(* IEC 61131-3 sources: rk/stdlib (part 3) *)

(* ---- Math.st ---- *)
/*
Arithmetic functions.

Each function has one overload per type it applies to, and returns the type
it was given. Angles are in radians.

A `REAL` or `LREAL` result follows IEEE 754: outside a function's domain it
is NaN, and at a pole it is infinite. Neither stops the scan. Test for them
with [Std.Math.IS_NAN] and [Std.Math.NOT_OK] where it matters.
*/
NAMESPACE Std.Math

	/* Returns the absolute value of `IN`, which is `IN` itself on an unsigned type.

	   The most negative value of a signed integer type has no positive
	   counterpart, and is returned as it is: `ABS(SINT#-128)` is -128.

	   # Examples

	   ```iecst
	   n := ABS(-5);    // 5
	   r := ABS(-2.5);  // 2.5
	   ```
	*/
	FUNCTION ABS: SINT
		VAR_INPUT
			IN: SINT
		END_VAR
		{wasm IN 'abs' (params IN) (result ABS)}
	END_FUNCTION

	FUNCTION ABS: INT
		VAR_INPUT
			IN: INT
		END_VAR
		{wasm IN 'abs' (params IN) (result ABS)}
	END_FUNCTION

	FUNCTION ABS: DINT
		VAR_INPUT
			IN: DINT
		END_VAR
		{wasm IN 'abs' (params IN) (result ABS)}
	END_FUNCTION

	FUNCTION ABS: LINT
		VAR_INPUT
			IN: LINT
		END_VAR
		{wasm IN 'abs' (params IN) (result ABS)}
	END_FUNCTION

	FUNCTION ABS: REAL
		VAR_INPUT
			IN: REAL
		END_VAR
		{wasm IN 'abs' (params IN) (result ABS)}
	END_FUNCTION

	FUNCTION ABS: LREAL
		VAR_INPUT
			IN: LREAL
		END_VAR
		{wasm IN 'abs' (params IN) (result ABS)}
	END_FUNCTION

	FUNCTION ABS: USINT
		VAR_INPUT
			IN: USINT
		END_VAR
		ABS := IN;
	END_FUNCTION

	FUNCTION ABS: UINT
		VAR_INPUT
			IN: UINT
		END_VAR
		ABS := IN;
	END_FUNCTION

	FUNCTION ABS: UDINT
		VAR_INPUT
			IN: UDINT
		END_VAR
		ABS := IN;
	END_FUNCTION

	FUNCTION ABS: ULINT
		VAR_INPUT
			IN: ULINT
		END_VAR
		ABS := IN;
	END_FUNCTION

	/* Returns the square root of `IN`.

	   Returns NaN when `IN` is negative.

	   # Examples

	   ```iecst
	   r := SQRT(9.0);  // 3.0
	   r := SQRT(2.0);  // 1.4142135
	   ```
	*/
	FUNCTION SQRT: REAL
		VAR_INPUT
			IN: REAL
		END_VAR
		{wasm IN 'sqrt' (params IN) (result SQRT)}
	END_FUNCTION

	FUNCTION SQRT: LREAL
		VAR_INPUT
			IN: LREAL
		END_VAR
		{wasm IN 'sqrt' (params IN) (result SQRT)}
	END_FUNCTION

	/* Returns the natural logarithm of `IN`.

	   Returns NaN when `IN` is negative, and negative infinity when it is 0.

	   # Examples

	   ```iecst
	   r := LN(1.0);  // 0.0
	   r := LN(2.0);  // 0.6931472
	   ```
	*/
	FUNCTION LN: REAL
		VAR_INPUT
			IN: REAL
		END_VAR
		{wasm IN 'ln' (params IN) (result LN)}
	END_FUNCTION

	FUNCTION LN: LREAL
		VAR_INPUT
			IN: LREAL
		END_VAR
		{wasm IN 'ln' (params IN) (result LN)}
	END_FUNCTION

	/* Returns the base 10 logarithm of `IN`.

	   Returns NaN when `IN` is negative, and negative infinity when it is 0.

	   # Examples

	   ```iecst
	   r := LOG(100.0);   // 2.0
	   r := LOG(1000.0);  // 3.0
	   ```
	*/
	FUNCTION LOG: REAL
		VAR_INPUT
			IN: REAL
		END_VAR
		{wasm IN 'log' (params IN) (result LOG)}
	END_FUNCTION

	FUNCTION LOG: LREAL
		VAR_INPUT
			IN: LREAL
		END_VAR
		{wasm IN 'log' (params IN) (result LOG)}
	END_FUNCTION

	/* Returns e raised to the power of `IN`.

	   # Examples

	   ```iecst
	   r := EXP(0.0);  // 1.0
	   r := EXP(1.0);  // 2.7182817
	   ```
	*/
	FUNCTION EXP: REAL
		VAR_INPUT
			IN: REAL
		END_VAR
		{wasm IN 'exp' (params IN) (result EXP)}
	END_FUNCTION

	FUNCTION EXP: LREAL
		VAR_INPUT
			IN: LREAL
		END_VAR
		{wasm IN 'exp' (params IN) (result EXP)}
	END_FUNCTION

	/* Returns the sine of `IN`, an angle in radians.

	   # Examples

	   ```iecst
	   r := SIN(0.0);  // 0.0
	   r := SIN(0.5);  // 0.4794255
	   ```
	*/
	FUNCTION SIN: REAL
		VAR_INPUT
			IN: REAL
		END_VAR
		{wasm IN 'sin' (params IN) (result SIN)}
	END_FUNCTION

	FUNCTION SIN: LREAL
		VAR_INPUT
			IN: LREAL
		END_VAR
		{wasm IN 'sin' (params IN) (result SIN)}
	END_FUNCTION

	/* Returns the cosine of `IN`, an angle in radians.

	   # Examples

	   ```iecst
	   r := COS(0.0);  // 1.0
	   r := COS(1.0);  // 0.5403023
	   ```
	*/
	FUNCTION COS: REAL
		VAR_INPUT
			IN: REAL
		END_VAR
		{wasm IN 'cos' (params IN) (result COS)}
	END_FUNCTION

	FUNCTION COS: LREAL
		VAR_INPUT
			IN: LREAL
		END_VAR
		{wasm IN 'cos' (params IN) (result COS)}
	END_FUNCTION

	/* Returns the tangent of `IN`, an angle in radians.

	   # Examples

	   ```iecst
	   r := TAN(0.0);  // 0.0
	   r := TAN(1.0);  // 1.5574077
	   ```
	*/
	FUNCTION TAN: REAL
		VAR_INPUT
			IN: REAL
		END_VAR
		{wasm IN 'tan' (params IN) (result TAN)}
	END_FUNCTION

	FUNCTION TAN: LREAL
		VAR_INPUT
			IN: LREAL
		END_VAR
		{wasm IN 'tan' (params IN) (result TAN)}
	END_FUNCTION

	/* Returns the arc sine of `IN`, in radians.

	   Returns NaN when `IN` is outside -1.0 to 1.0.

	   # Examples

	   ```iecst
	   r := ASIN(0.0);  // 0.0
	   r := ASIN(1.0);  // 1.5707964
	   ```
	*/
	FUNCTION ASIN: REAL
		VAR_INPUT
			IN: REAL
		END_VAR
		{wasm IN 'asin' (params IN) (result ASIN)}
	END_FUNCTION

	FUNCTION ASIN: LREAL
		VAR_INPUT
			IN: LREAL
		END_VAR
		{wasm IN 'asin' (params IN) (result ASIN)}
	END_FUNCTION

	/* Returns the arc cosine of `IN`, in radians.

	   Returns NaN when `IN` is outside -1.0 to 1.0.

	   # Examples

	   ```iecst
	   r := ACOS(1.0);  // 0.0
	   r := ACOS(0.0);  // 1.5707964
	   ```
	*/
	FUNCTION ACOS: REAL
		VAR_INPUT
			IN: REAL
		END_VAR
		{wasm IN 'acos' (params IN) (result ACOS)}
	END_FUNCTION

	FUNCTION ACOS: LREAL
		VAR_INPUT
			IN: LREAL
		END_VAR
		{wasm IN 'acos' (params IN) (result ACOS)}
	END_FUNCTION

	/* Returns the arc tangent of `IN`, in radians.

	   # Examples

	   ```iecst
	   r := ATAN(0.0);  // 0.0
	   r := ATAN(1.0);  // 0.7853982
	   ```
	*/
	FUNCTION ATAN: REAL
		VAR_INPUT
			IN: REAL
		END_VAR
		{wasm IN 'atan' (params IN) (result ATAN)}
	END_FUNCTION

	FUNCTION ATAN: LREAL
		VAR_INPUT
			IN: LREAL
		END_VAR
		{wasm IN 'atan' (params IN) (result ATAN)}
	END_FUNCTION

	/* Returns the angle of the point (`X`, `Y`), in radians.

	   This is the arc tangent of `IN / IN2`, with the signs of both used to pick
	   the quadrant. `Y` is the y coordinate and `X` the x.

	   # Examples

	   ```iecst
	   r := ATAN2(1.0, 1.0);    // 0.7853982
	   r := ATAN2(1.0, -1.0);   // 2.3561945
	   r := ATAN2(-1.0, 1.0);   // -0.7853982
	   ```
	*/
	FUNCTION ATAN2: REAL
		VAR_INPUT
			Y: REAL
			X: REAL
		END_VAR
		{wasm Y 'atan2' (params Y X) (result ATAN2)}
	END_FUNCTION

	FUNCTION ATAN2: LREAL
		VAR_INPUT
			Y: LREAL
			X: LREAL
		END_VAR
		{wasm Y 'atan2' (params Y X) (result ATAN2)}
	END_FUNCTION

	/* Returns `IN1` raised to the power of `IN2`.

	   This is the `**` operator as a function. `IN2` may be an integer, and the
	   result has the type of `IN1`.

	   # Examples

	   ```iecst
	   r := EXPT(2.0, 3.0);  // 8.0
	   r := EXPT(9.0, 0.5);  // 3.0
	   ```
	*/
	FUNCTION EXPT: REAL
		VAR_INPUT
			IN1: REAL
			IN2: REAL
		END_VAR
		{wasm IN1 'pow' (params IN1 IN2) (result EXPT)}
	END_FUNCTION

	FUNCTION EXPT: LREAL
		VAR_INPUT
			IN1: LREAL
			IN2: LREAL
		END_VAR
		{wasm IN1 'pow' (params IN1 IN2) (result EXPT)}
	END_FUNCTION

	FUNCTION EXPT: REAL
		VAR_INPUT
			IN1: REAL
			IN2: LREAL
		END_VAR
		EXPT := IN1 ** IN2;
	END_FUNCTION

	FUNCTION EXPT: REAL
		VAR_INPUT
			IN1: REAL
			IN2: SINT
		END_VAR
		EXPT := IN1 ** IN2;
	END_FUNCTION

	FUNCTION EXPT: REAL
		VAR_INPUT
			IN1: REAL
			IN2: INT
		END_VAR
		EXPT := IN1 ** IN2;
	END_FUNCTION

	FUNCTION EXPT: REAL
		VAR_INPUT
			IN1: REAL
			IN2: DINT
		END_VAR
		EXPT := IN1 ** IN2;
	END_FUNCTION

	FUNCTION EXPT: REAL
		VAR_INPUT
			IN1: REAL
			IN2: LINT
		END_VAR
		EXPT := IN1 ** IN2;
	END_FUNCTION

	FUNCTION EXPT: REAL
		VAR_INPUT
			IN1: REAL
			IN2: USINT
		END_VAR
		EXPT := IN1 ** IN2;
	END_FUNCTION

	FUNCTION EXPT: REAL
		VAR_INPUT
			IN1: REAL
			IN2: UINT
		END_VAR
		EXPT := IN1 ** IN2;
	END_FUNCTION

	FUNCTION EXPT: REAL
		VAR_INPUT
			IN1: REAL
			IN2: UDINT
		END_VAR
		EXPT := IN1 ** IN2;
	END_FUNCTION

	FUNCTION EXPT: REAL
		VAR_INPUT
			IN1: REAL
			IN2: ULINT
		END_VAR
		EXPT := IN1 ** IN2;
	END_FUNCTION

	FUNCTION EXPT: LREAL
		VAR_INPUT
			IN1: LREAL
			IN2: REAL
		END_VAR
		EXPT := IN1 ** IN2;
	END_FUNCTION

	FUNCTION EXPT: LREAL
		VAR_INPUT
			IN1: LREAL
			IN2: SINT
		END_VAR
		EXPT := IN1 ** IN2;
	END_FUNCTION

	FUNCTION EXPT: LREAL
		VAR_INPUT
			IN1: LREAL
			IN2: INT
		END_VAR
		EXPT := IN1 ** IN2;
	END_FUNCTION

	FUNCTION EXPT: LREAL
		VAR_INPUT
			IN1: LREAL
			IN2: DINT
		END_VAR
		EXPT := IN1 ** IN2;
	END_FUNCTION

	FUNCTION EXPT: LREAL
		VAR_INPUT
			IN1: LREAL
			IN2: LINT
		END_VAR
		EXPT := IN1 ** IN2;
	END_FUNCTION

	FUNCTION EXPT: LREAL
		VAR_INPUT
			IN1: LREAL
			IN2: USINT
		END_VAR
		EXPT := IN1 ** IN2;
	END_FUNCTION

	FUNCTION EXPT: LREAL
		VAR_INPUT
			IN1: LREAL
			IN2: UINT
		END_VAR
		EXPT := IN1 ** IN2;
	END_FUNCTION

	FUNCTION EXPT: LREAL
		VAR_INPUT
			IN1: LREAL
			IN2: UDINT
		END_VAR
		EXPT := IN1 ** IN2;
	END_FUNCTION

	FUNCTION EXPT: LREAL
		VAR_INPUT
			IN1: LREAL
			IN2: ULINT
		END_VAR
		EXPT := IN1 ** IN2;
	END_FUNCTION

	/* Returns `TRUE` if `IN` is not a number.

	   NaN comes from `0.0 / 0.0`, from the square root of a negative, and above
	   all from a bit pattern read off a fieldbus or an analog channel. It spreads
	   through arithmetic and converts to 0, so test for it where it matters.

	   See [Std.Math.NOT_OK] to refuse an infinite value as well.
	*/
	FUNCTION IS_NAN: BOOL
		VAR_INPUT
			IN: REAL;
		END_VAR
		IS_NAN := IN <> IN;
	END_FUNCTION

	FUNCTION IS_NAN: BOOL
		VAR_INPUT
			IN: LREAL;
		END_VAR
		IS_NAN := IN <> IN;
	END_FUNCTION

	/* Returns `TRUE` if `IN` is not a number, or is infinite.

	   # Examples

	   ```iecst
	   IF NOT_OK(measured) THEN
	       alarm := TRUE;
	   END_IF;
	   ```
	*/
	FUNCTION NOT_OK: BOOL
		VAR_INPUT
			IN: REAL;
		END_VAR
		NOT_OK := (IN - IN) <> 0.0;
	END_FUNCTION

	FUNCTION NOT_OK: BOOL
		VAR_INPUT
			IN: LREAL;
		END_VAR
		NOT_OK := (IN - IN) <> LREAL#0.0;
	END_FUNCTION

	NAMESPACE Test
		USING Std.Unit

		// ----- EXPT ---------------------------------------------------
		{test}
		FUNCTION test_is_nan
			VAR
				z: REAL := 0.0;
			END_VAR
			ASSERT(IS_NAN(z / z) AND NOT IS_NAN(1.5) AND NOT IS_NAN(1.0 / z));
		END_FUNCTION

		{test}
		FUNCTION test_not_ok_is_nan_or_infinite
			VAR
				z: REAL := 0.0;
			END_VAR
			ASSERT(NOT_OK(z / z) AND NOT_OK(1.0 / z) AND NOT_OK(-1.0 / z) AND NOT NOT_OK(3.0));
		END_FUNCTION

		{test}
		FUNCTION test_expt_real ASSERT(EXPT(2.0, 3.0) = 8.0);
		END_FUNCTION

		{test}
		FUNCTION test_expt_fractional ASSERT(EXPT(9.0, 0.5) = 3.0);
		END_FUNCTION

		// The result has the type of IN1, whatever the exponent's: a REAL
		// raised to a DINT is stored in a REAL, which an LREAL result is not.
		{test}
		FUNCTION test_expt_keeps_the_base_type
		VAR r: REAL; l: LREAL; n: DINT := 3; u: USINT := 10; END_VAR
			r := EXPT(REAL#2.0, n);
			ASSERT(r = 8.0);
			r := EXPT(REAL#2.0, LREAL#0.5);
			ASSERT(r > 1.41 AND r < 1.42);
			l := EXPT(LREAL#2.0, u);
			ASSERT(l = LREAL#1024.0);
		END_FUNCTION

		{test}
		FUNCTION test_expt_integer_exponent
		VAR x: REAL; n: INT; END_VAR
			x := 2.0;
			n := 10;
			ASSERT(EXPT(x, n) = 1024.0);
		END_FUNCTION

		{test}
		FUNCTION test_expt_lreal ASSERT(EXPT(LREAL#2.0, LREAL#10.0) = LREAL#1024.0);
		END_FUNCTION

		// The result has the type of IN1, whatever the exponent: a REAL target
		// refuses an LREAL.
		{test}
		FUNCTION test_expt_keeps_the_type_of_in1
			VAR
				r: REAL := 2.0;
				l: LREAL := 2.0;
				a: REAL;
				b: LREAL;
				si: SINT := 3;
				i: INT := 3;
				d: DINT := 3;
				n: LINT := 3;
				us: USINT := 3;
				u: UINT := 3;
				ud: UDINT := 3;
				ul: ULINT := 3;
				x: REAL := 3.0;
				y: LREAL := 3.0;
			END_VAR
			a := EXPT(r, si); ASSERT(a = 8.0);
			a := EXPT(r, i); ASSERT(a = 8.0);
			a := EXPT(r, d); ASSERT(a = 8.0);
			a := EXPT(r, n); ASSERT(a = 8.0);
			a := EXPT(r, us); ASSERT(a = 8.0);
			a := EXPT(r, u); ASSERT(a = 8.0);
			a := EXPT(r, ud); ASSERT(a = 8.0);
			a := EXPT(r, ul); ASSERT(a = 8.0);
			a := EXPT(r, x); ASSERT(a = 8.0);
			a := EXPT(r, y); ASSERT(a = 8.0);
			b := EXPT(l, si); ASSERT(b = LREAL#8.0);
			b := EXPT(l, i); ASSERT(b = LREAL#8.0);
			b := EXPT(l, d); ASSERT(b = LREAL#8.0);
			b := EXPT(l, n); ASSERT(b = LREAL#8.0);
			b := EXPT(l, us); ASSERT(b = LREAL#8.0);
			b := EXPT(l, u); ASSERT(b = LREAL#8.0);
			b := EXPT(l, ud); ASSERT(b = LREAL#8.0);
			b := EXPT(l, ul); ASSERT(b = LREAL#8.0);
			b := EXPT(l, x); ASSERT(b = LREAL#8.0);
			b := EXPT(l, y); ASSERT(b = LREAL#8.0);
		END_FUNCTION

		{test}
		FUNCTION test_expt_takes_literals
			VAR
				r: REAL := 2.0;
				l: LREAL := 2.0;
				a: REAL;
				b: LREAL;
			END_VAR
			a := EXPT(2.0, 3.0); ASSERT(a = 8.0);
			a := EXPT(r, 3.0); ASSERT(a = 8.0);
			a := EXPT(r, 3); ASSERT(a = 8.0);
			a := EXPT(2.0, 3); ASSERT(a = 8.0);
			a := EXPT(r, DINT#3); ASSERT(a = 8.0);
			a := EXPT(IN1 := r, IN2 := 3); ASSERT(a = 8.0);
			b := EXPT(l, 3); ASSERT(b = LREAL#8.0);
			b := EXPT(l, 3.0); ASSERT(b = LREAL#8.0);
			b := EXPT(LREAL#2.0, 3); ASSERT(b = LREAL#8.0);
			b := EXPT(l, -1); ASSERT(b = LREAL#0.5);
		END_FUNCTION

		{test}
		FUNCTION test_abs_of_an_unsigned_is_itself
			VAR
				us: USINT := 200;
				u: UINT := 60000;
				ud: UDINT := 4000000000;
				ul: ULINT := 18446744073709551615;
			END_VAR
			us := ABS(us); ASSERT(us = 200);
			u := ABS(u); ASSERT(u = 60000);
			ud := ABS(ud); ASSERT(ud = 4000000000);
			ul := ABS(ul); ASSERT(ul = 18446744073709551615);
		END_FUNCTION

		{test}
		FUNCTION test_expt_matches_operator
		VAR x: REAL; END_VAR
			x := 3.0;
			ASSERT(EXPT(x, 2.0) = x ** 2.0);
		END_FUNCTION

		// ----- ABS (per signed-numeric overloads) ---------------------
		{test}
		FUNCTION test_abs_positive ASSERT(ABS(5) = 5);
		END_FUNCTION

		{test}
		FUNCTION test_abs_negative ASSERT(ABS(-42) = 42);
		END_FUNCTION

		{test}
		FUNCTION test_abs_zero ASSERT(ABS(0) = 0);
		END_FUNCTION

		{test}
		FUNCTION test_abs_real ASSERT(ABS(-2.5) = 2.5);
		END_FUNCTION

		{test}
		FUNCTION test_abs_real_positive ASSERT(ABS(3.14) = 3.14);
		END_FUNCTION

		{test}
		FUNCTION test_abs_with_message ASSERT(ABS(-7) = 7, 'ABS should return the positive value');
		END_FUNCTION

		// An unsigned value is its own absolute value, the largest included.
		{test}
		FUNCTION test_abs_unsigned
			ASSERT(ABS(USINT#255) = USINT#255);
			ASSERT(ABS(UINT#65535) = UINT#65535);
			ASSERT(ABS(UDINT#4294967295) = UDINT#4294967295);
			ASSERT(ABS(ULINT#18446744073709551615) = ULINT#18446744073709551615);
		END_FUNCTION

		// ----- SQRT (REAL/LREAL overloads) ----------------------------
		{test}
		FUNCTION test_sqrt_9 ASSERT(SQRT(9.0) = 3.0);
		END_FUNCTION

		{test}
		FUNCTION test_sqrt_4 ASSERT(SQRT(4.0) = 2.0);
		END_FUNCTION

		{test}
		FUNCTION test_sqrt_1 ASSERT(SQRT(1.0) = 1.0);
		END_FUNCTION

		// ----- Trigonometric (REAL/LREAL overloads) -------------------
		{test}
		FUNCTION test_sin_zero ASSERT(SIN(0.0) = 0.0);
		END_FUNCTION

		{test}
		FUNCTION test_cos_zero ASSERT(COS(0.0) = 1.0);
		END_FUNCTION

		{test}
		FUNCTION test_tan_zero ASSERT(TAN(0.0) = 0.0);
		END_FUNCTION

		{test}
		FUNCTION test_asin_zero ASSERT(ASIN(0.0) = 0.0);
		END_FUNCTION

		{test}
		FUNCTION test_acos_one ASSERT(ACOS(1.0) = 0.0);
		END_FUNCTION

		{test}
		FUNCTION test_atan_zero ASSERT(ATAN(0.0) = 0.0);
		END_FUNCTION

		// ----- Logarithmic / Exponential (REAL/LREAL overloads) ------
		{test}
		FUNCTION test_ln_1 ASSERT(LN(1.0) = 0.0);
		END_FUNCTION

		{test}
		FUNCTION test_log_1 ASSERT(LOG(1.0) = 0.0);
		END_FUNCTION

		{test}
		FUNCTION test_exp_0 ASSERT(EXP(0.0) = 1.0);
		END_FUNCTION

		// ----- Arithmetic operators --------------------------------------------------------------------------------
		{test}
		FUNCTION test_add_int
			VAR
				r: INT;
			END_VAR
			r := 3 + 4;
			ASSERT(r = 7);
		END_FUNCTION

		{test}
		FUNCTION test_sub_int
			VAR
				r: INT;
			END_VAR
			r := 10 - 3;
			ASSERT(r = 7);
		END_FUNCTION

		{test}
		FUNCTION test_mul_int
			VAR
				r: INT;
			END_VAR
			r := 6 * 7;
			ASSERT(r = 42);
		END_FUNCTION

		{test}
		FUNCTION test_div_int
			VAR
				r: INT;
			END_VAR
			r := 100 / 10;
			ASSERT(r = 10);
		END_FUNCTION

		{test}
		FUNCTION test_mod_int
			VAR
				r: INT;
			END_VAR
			r := 10 MOD 3;
			ASSERT(r = 1);
		END_FUNCTION

		{test}
		FUNCTION test_add_real
			VAR
				r: REAL;
			END_VAR
			r := 1.5 + 2.5;
			ASSERT(r = 4.0);
		END_FUNCTION

		{test}
		FUNCTION test_sub_negative
			VAR
				r: INT;
			END_VAR
			r := 3 - 10;
			ASSERT(r = -7);
		END_FUNCTION

		{test}
		FUNCTION test_nested_arithmetic
			VAR
				a: INT;
				b: INT;
				c: INT;
			END_VAR
			a := 2 * 3;
			b := 4 * 5;
			c := a + b;
			ASSERT(c = 26);
		END_FUNCTION

		// ----- Variable assignment ---------------------------------------------------------------------------------
		{test}
		FUNCTION test_var_assignment
			VAR
				x: INT := 10;
				y: INT;
			END_VAR
			y := x;
			ASSERT(x = y);
		END_FUNCTION

		{test}
		FUNCTION test_var_init
			VAR
				x: INT := 42;
			END_VAR
			ASSERT(x = 42);
		END_FUNCTION

		{test}
		FUNCTION test_var_default_zero
			VAR
				x: INT;
			END_VAR
			ASSERT(x = 0);
		END_FUNCTION

		{test}
		FUNCTION test_var_bool_init
			VAR
				b: BOOL := TRUE;
			END_VAR
			ASSERT(b);
		END_FUNCTION

		{test}
		FUNCTION test_var_real_init
			VAR
				r: REAL := 3.14;
			END_VAR
			ASSERT(r = 3.14);
		END_FUNCTION

		// ----- Boolean logic ---------------------------------------------------------------------------------------
		{test}
		FUNCTION test_bool_and_tt
			VAR
				a: BOOL := TRUE;
				b: BOOL := TRUE;
			END_VAR
			ASSERT(a AND b);
		END_FUNCTION

		{test}
		FUNCTION test_bool_and_tf
			VAR
				a: BOOL := TRUE;
				b: BOOL := FALSE;
			END_VAR
			ASSERT(NOT (a AND b));
		END_FUNCTION

		{test}
		FUNCTION test_bool_or_tf
			VAR
				a: BOOL := FALSE;
				b: BOOL := TRUE;
			END_VAR
			ASSERT(a OR b);
		END_FUNCTION

		{test}
		FUNCTION test_bool_or_ff
			VAR
				a: BOOL := FALSE;
				b: BOOL := FALSE;
			END_VAR
			ASSERT(NOT (a OR b));
		END_FUNCTION

		{test}
		FUNCTION test_bool_not
			VAR
				a: BOOL := FALSE;
			END_VAR
			ASSERT(NOT a);
		END_FUNCTION

		{test}
		FUNCTION test_bool_xor
			VAR
				a: BOOL := TRUE;
				b: BOOL := FALSE;
			END_VAR
			ASSERT(a XOR b);
		END_FUNCTION

		{test}
		FUNCTION test_bool_xor_same
			VAR
				a: BOOL := TRUE;
				b: BOOL := TRUE;
			END_VAR
			ASSERT(NOT (a XOR b));
		END_FUNCTION

		// ----- Comparison operators --------------------------------------------------------------------------------
		{test}
		FUNCTION test_cmp_eq
			VAR
				a: INT := 5;
			END_VAR
			ASSERT(a = 5);
		END_FUNCTION

		{test}
		FUNCTION test_cmp_ne
			VAR
				a: INT := 1;
				b: INT := 2;
			END_VAR
			ASSERT(a <> b);
		END_FUNCTION

		{test}
		FUNCTION test_cmp_lt
			VAR
				a: INT := 3;
				b: INT := 5;
			END_VAR
			ASSERT(a < b);
		END_FUNCTION

		{test}
		FUNCTION test_cmp_le
			VAR
				a: INT := 5;
			END_VAR
			ASSERT(a <= 5);
		END_FUNCTION

		{test}
		FUNCTION test_cmp_gt
			VAR
				a: INT := 10;
				b: INT := 5;
			END_VAR
			ASSERT(a > b);
		END_FUNCTION

		{test}
		FUNCTION test_cmp_ge
			VAR
				a: INT := 5;
			END_VAR
			ASSERT(a >= 5);
		END_FUNCTION

		// ----- Control flow: IF ------------------------------------------------------------------------------------
		{test}
		FUNCTION test_if_true
			VAR
				r: INT := 0;
			END_VAR
			IF TRUE THEN
				r := 1;
			END_IF;
			ASSERT(r = 1);
		END_FUNCTION

		{test}
		FUNCTION test_if_false
			VAR
				r: INT := 0;
			END_VAR
			IF FALSE THEN
				r := 1;
			END_IF;
			ASSERT(r = 0);
		END_FUNCTION

		{test}
		FUNCTION test_if_else
			VAR
				r: INT := 0;
			END_VAR
			IF FALSE THEN
				r := 1;
			ELSE
				r := 2;
			END_IF;
			ASSERT(r = 2);
		END_FUNCTION

		{test}
		FUNCTION test_if_elsif
			VAR
				r: INT := 0;
				x: INT := 2;
			END_VAR
			IF x = 1 THEN
				r := 10;
			ELSIF x = 2 THEN
				r := 20;
			ELSE
				r := 30;
			END_IF;
			ASSERT(r = 20);
		END_FUNCTION

		// ----- Control flow: FOR -----------------------------------------------------------------------------------
		{test}
		FUNCTION test_for_sum
			VAR
				sum: INT := 0;
				i: INT;
			END_VAR
			FOR i := 1 TO 5 DO
				sum := sum + i;
			END_FOR;
			ASSERT(sum = 15);
		END_FUNCTION

		{test}
		FUNCTION test_for_single
			VAR
				r: INT := 0;
				i: INT;
			END_VAR
			FOR i := 5 TO 5 DO
				r := r + 1;
			END_FOR;
			ASSERT(r = 1);
		END_FUNCTION

		{test}
		FUNCTION test_for_descending
			VAR
				n: INT := 0;
				i: INT;
			END_VAR
			// A constant negative BY flips the exit comparison: this loop
			// used to exit before its first iteration.
			FOR i := 10 TO 1 BY -1 DO
				n := n + 1;
			END_FOR;
			ASSERT(n = 10, 'descending FOR runs all 10 iterations');
		END_FUNCTION

		{test}
		FUNCTION test_for_lint_counter
			VAR
				n: LINT := 0;
				i: LINT;
			END_VAR
			// i64-lane control variable (used to emit invalid wasm).
			FOR i := LINT#1 TO LINT#3 DO
				n := n + i;
			END_FOR;
			ASSERT(n = LINT#6, 'LINT FOR loop sums 1+2+3');
		END_FUNCTION

		{test}
		FUNCTION test_for_lint_descending_beyond_i32
			VAR
				n: LINT := 0;
				i: LINT;
			END_VAR
			FOR i := LINT#5000000002 TO LINT#5000000000 BY LINT#-1 DO
				n := n + 1;
			END_FOR;
			ASSERT(n = LINT#3, 'descending i64 FOR with bounds beyond i32 range');
		END_FUNCTION

		{test}
		FUNCTION test_for_subwidth_counter_stays_in_domain
			VAR
				n: USINT := 0;
				i: USINT;
			END_VAR
			// Counter increments stay in the type's domain. NOTE: an upper
			// bound at the type MAX (e.g. TO 255) wraps before the exit
			// check and never terminates; keep bounds below the type maximum.
			FOR i := 250 TO 254 DO
				n := n + 1;
			END_FOR;
			ASSERT(n = USINT#5, 'body ran 5 times');
			{allow 'loop-var-after-loop'}
			ASSERT(i = USINT#255, 'counter exits in-domain at 255');
		END_FUNCTION

		// ----- Control flow: WHILE ---------------------------------------------------------------------------------
		{test}
		FUNCTION test_while_count
			VAR
				count: INT := 0;
			END_VAR
			WHILE count < 10 DO
				count := count + 1;
			END_WHILE;
			ASSERT(count = 10);
		END_FUNCTION

		{test}
		FUNCTION test_while_false
			VAR
				count: INT := 0;
			END_VAR
			WHILE FALSE DO
				count := count + 1;
			END_WHILE;
			ASSERT(count = 0);
		END_FUNCTION

		// ----- Control flow: REPEAT --------------------------------------------------------------------------------
		{test}
		FUNCTION test_repeat_until
			VAR
				count: INT := 0;
			END_VAR
			REPEAT count := count + 1;
				UNTIL count >= 5
			END_REPEAT;
			ASSERT(count = 5);
		END_FUNCTION

		// ----- Function calls with return values ----------------------
		{test}
		FUNCTION test_func_return
			VAR
				r: INT;
			END_VAR
			r := ABS(-99);
			ASSERT(r = 99);
		END_FUNCTION

		// Chained calls via intermediate variable
		{test}
		FUNCTION test_chained_abs
			VAR
				inner: INT;
				r: INT;
			END_VAR
			inner := ABS(-5);
			r := ABS(inner);
			ASSERT(r = 5);
		END_FUNCTION

		// ----- Type widths -----------------------------------------------------------------------------------------
		{test}
		FUNCTION test_lint_arithmetic
			VAR
				a: LINT := 1000000000;
				b: LINT := 2000000000;
				c: LINT;
			END_VAR
			c := a + b;
			ASSERT(c = 3000000000);
		END_FUNCTION

		{test}
		FUNCTION test_lreal_precision
			VAR
				a: LREAL := 1.0;
				b: LREAL := 3.0;
				c: LREAL;
			END_VAR
			c := a / b;
			// Can't compare exactly, but c * 3.0 should be 1.0
			ASSERT(c * b = a);
		END_FUNCTION

		// --- transcendentals at nonzero, non-colliding points: the fixed
		// points used above (0->0, 1->0, 0->1) are shared across the whole
		// family, so swapped imports (ln vs log, exp vs cos) pass unnoticed ---

		{test}
		FUNCTION test_trig_nonzero_points_real
			ASSERT(ABS(SIN(0.5) - 0.4794255) < 0.0001, 'SIN(0.5)');
			ASSERT(ABS(COS(1.0) - 0.5403023) < 0.0001, 'COS(1.0)');
			ASSERT(ABS(TAN(1.0) - 1.5574077) < 0.0001, 'TAN(1.0)');
			ASSERT(ABS(ASIN(0.5) - 0.5235988) < 0.0001, 'ASIN(0.5) = pi/6');
			ASSERT(ABS(ACOS(0.5) - 1.0471976) < 0.0001, 'ACOS(0.5) = pi/3');
			ASSERT(ABS(ATAN(1.0) - 0.7853982) < 0.0001, 'ATAN(1.0) = pi/4');
		END_FUNCTION

		{test}
		FUNCTION test_trig_nonzero_points_lreal
			ASSERT(ABS(SIN(LREAL#0.5) - LREAL#0.479425538604203) < LREAL#0.000000001, 'SIN LREAL');
			ASSERT(ABS(COS(LREAL#1.0) - LREAL#0.540302305868140) < LREAL#0.000000001, 'COS LREAL');
			ASSERT(ABS(ATAN(LREAL#1.0) - LREAL#0.785398163397448) < LREAL#0.000000001, 'ATAN LREAL = pi/4');
		END_FUNCTION

		{test}
		FUNCTION test_log_exp_nonzero_points
			ASSERT(ABS(LN(2.0) - 0.6931472) < 0.0001, 'LN(2)');
			ASSERT(ABS(LOG(100.0) - 2.0) < 0.0001, 'LOG(100) = 2, distinguishes LOG from LN');
			ASSERT(ABS(EXP(1.0) - 2.7182818) < 0.0001, 'EXP(1) = e');
			ASSERT(ABS(SQRT(2.0) - 1.4142136) < 0.0001, 'SQRT(2)');
			ASSERT(ABS(LN(LREAL#2.0) - LREAL#0.693147180559945) < LREAL#0.000000001, 'LN LREAL');
			ASSERT(ABS(EXP(LREAL#1.0) - LREAL#2.718281828459045) < LREAL#0.000000001, 'EXP LREAL');
			ASSERT(ABS(LOG(LREAL#1000.0) - LREAL#3.0) < LREAL#0.000000001, 'LOG LREAL');
			ASSERT(ABS(SQRT(LREAL#2.0) - LREAL#1.414213562373095) < LREAL#0.000000001, 'SQRT LREAL');
		END_FUNCTION

		// --- ATAN2: the one two-argument function. Swapped y/x is only
		// detectable with an asymmetric quadrant pair ---

		{test}
		FUNCTION test_atan2_quadrants_real
			ASSERT(ABS(ATAN2(1.0, -1.0) - 2.3561945) < 0.0001, 'ATAN2(+y,-x) = 3pi/4 (2nd quadrant)');
			ASSERT(ABS(ATAN2(-1.0, 1.0) - (-0.7853982)) < 0.0001, 'ATAN2(-y,+x) = -pi/4 (4th quadrant)');
		END_FUNCTION

		{test}
		FUNCTION test_atan2_quadrants_lreal
			ASSERT(ABS(ATAN2(LREAL#1.0, LREAL#-1.0) - LREAL#2.356194490192345) < LREAL#0.000000001, 'ATAN2 LREAL 3pi/4');
			ASSERT(ABS(ATAN2(LREAL#-1.0, LREAL#1.0) - LREAL#-0.785398163397448) < LREAL#0.000000001, 'ATAN2 LREAL -pi/4');
		END_FUNCTION

		// --- ABS boundaries and the dark overloads ---

		{test}
		FUNCTION test_abs_boundaries
			ASSERT_EQ(ABS(SINT#-127), SINT#127, 'ABS SINT near MIN');
			ASSERT_EQ(ABS(INT#-32767), INT#32767, 'ABS INT near MIN');
			ASSERT_EQ(ABS(DINT#-2147483647), DINT#2147483647, 'ABS DINT near MIN');
			ASSERT_EQ(ABS(LINT#-5000000000), LINT#5000000000, 'ABS LINT on the i64 lane');
		END_FUNCTION

		// --- sub-width integer arithmetic wraps at the IEC type width.
		// Values must never escape the type's domain ---

		{test}
		FUNCTION test_subwidth_arithmetic_wraps
			VAR
				a: USINT := 255;
				b: USINT := 1;
				z: USINT := 0;
				m: USINT := 16;
				i: INT := 32767;
				one: INT := 1;
				imin: INT := -32768;
				u16a: UINT := 65535;
			END_VAR
			ASSERT(a + b = USINT#0, 'USINT 255+1 wraps to 0');
			ASSERT(z - b = USINT#255, 'USINT 0-1 wraps to 255');
			ASSERT(m * m = USINT#0, 'USINT 16*16 wraps to 0');
			ASSERT(i + one = INT#-32768, 'INT 32767+1 wraps to -32768');
			ASSERT(imin - one = INT#32767, 'INT -32768-1 wraps to 32767');
			ASSERT(u16a * u16a = UINT#1, 'UINT 65535*65535 wraps to 1');
		END_FUNCTION

		{test}
		FUNCTION test_subwidth_negation_wraps
			VAR
				s: SINT := -128;
				sm1: SINT := -1;
			END_VAR
			ASSERT(-s = SINT#-128, 'NEG(SINT#-128) wraps to -128');
			ASSERT(s / sm1 = SINT#-128, 'SINT -128/-1 wraps to -128');
			ASSERT(ABS(s) = SINT#-128, 'ABS(SINT#-128) wraps to -128');
			ASSERT(ABS(SINT#-127) = SINT#127, 'ABS in-range is unaffected');
		END_FUNCTION

		// --- domain edges (pins current IEEE 754 behavior through libm) ---

		{test}
		FUNCTION test_float_domain_edges_pin_current
			(* pins current behavior: IEEE semantics, NaN for out-of-domain,
			   infinities at the poles. NaN is the only value with x <> x. *)
			ASSERT(SQRT(-1.0) <> SQRT(-1.0), 'SQRT(-1) is NaN');
			ASSERT(LN(-1.0) <> LN(-1.0), 'LN(-1) is NaN');
			ASSERT(LN(0.0) < -1000000.0, 'LN(0) is -inf');
			ASSERT(EXP(1000.0) > 1000000.0, 'EXP(1000) overflows to +inf');
		END_FUNCTION

		// wasm traps on the minimum divided by -1; the compiler guards it, so
		// the quotient wraps like every other overflow.
		{test}
		FUNCTION test_division_at_the_minimum_wraps
			VAR i : INT := INT#-32768; d : DINT := DINT#-2147483648; l : LINT := -LINT#9223372036854775807 - LINT#1; END_VAR
			ASSERT(i / INT#-1 = INT#-32768, 'INT');
			ASSERT(d / DINT#-1 = DINT#-2147483648, 'DINT');
			ASSERT(l / LINT#-1 = l, 'LINT');
			ASSERT(d MOD DINT#-1 = DINT#0, 'MOD is 0');
		END_FUNCTION
	END_NAMESPACE
END_NAMESPACE

(* ---- Memory.st ---- *)
/*
Memory functions.
*/
NAMESPACE Std.Memory

	/* Returns `IN`, and copies it into `OUT`.

	   There is one overload per elementary type.

	   # Examples

	   ```iecst
	   x := MOVE(42);       // x is 42
	   MOVE(42, OUT => x);  // x is 42
	   ```
	*/
	FUNCTION MOVE: BOOL
		VAR_INPUT
			IN: BOOL;
		END_VAR
		VAR_OUTPUT
			OUT: BOOL;
		END_VAR

		OUT := IN;
		MOVE := IN;
	END_FUNCTION

	FUNCTION MOVE: SINT
		VAR_INPUT
			IN: SINT;
		END_VAR
		VAR_OUTPUT
			OUT: SINT;
		END_VAR

		OUT := IN;
		MOVE := IN;
	END_FUNCTION

	FUNCTION MOVE: INT
		VAR_INPUT
			IN: INT;
		END_VAR
		VAR_OUTPUT
			OUT: INT;
		END_VAR

		OUT := IN;
		MOVE := IN;
	END_FUNCTION

	FUNCTION MOVE: DINT
		VAR_INPUT
			IN: DINT;
		END_VAR
		VAR_OUTPUT
			OUT: DINT;
		END_VAR

		OUT := IN;
		MOVE := IN;
	END_FUNCTION

	FUNCTION MOVE: LINT
		VAR_INPUT
			IN: LINT;
		END_VAR
		VAR_OUTPUT
			OUT: LINT;
		END_VAR

		OUT := IN;
		MOVE := IN;
	END_FUNCTION

	FUNCTION MOVE: USINT
		VAR_INPUT
			IN: USINT;
		END_VAR
		VAR_OUTPUT
			OUT: USINT;
		END_VAR

		OUT := IN;
		MOVE := IN;
	END_FUNCTION

	FUNCTION MOVE: UINT
		VAR_INPUT
			IN: UINT;
		END_VAR
		VAR_OUTPUT
			OUT: UINT;
		END_VAR

		OUT := IN;
		MOVE := IN;
	END_FUNCTION

	FUNCTION MOVE: UDINT
		VAR_INPUT
			IN: UDINT;
		END_VAR
		VAR_OUTPUT
			OUT: UDINT;
		END_VAR

		OUT := IN;
		MOVE := IN;
	END_FUNCTION

	FUNCTION MOVE: ULINT
		VAR_INPUT
			IN: ULINT;
		END_VAR
		VAR_OUTPUT
			OUT: ULINT;
		END_VAR

		OUT := IN;
		MOVE := IN;
	END_FUNCTION

	FUNCTION MOVE: BYTE
		VAR_INPUT
			IN: BYTE;
		END_VAR
		VAR_OUTPUT
			OUT: BYTE;
		END_VAR

		OUT := IN;
		MOVE := IN;
	END_FUNCTION

	FUNCTION MOVE: WORD
		VAR_INPUT
			IN: WORD;
		END_VAR
		VAR_OUTPUT
			OUT: WORD;
		END_VAR

		OUT := IN;
		MOVE := IN;
	END_FUNCTION

	FUNCTION MOVE: DWORD
		VAR_INPUT
			IN: DWORD;
		END_VAR
		VAR_OUTPUT
			OUT: DWORD;
		END_VAR

		OUT := IN;
		MOVE := IN;
	END_FUNCTION

	FUNCTION MOVE: LWORD
		VAR_INPUT
			IN: LWORD;
		END_VAR
		VAR_OUTPUT
			OUT: LWORD;
		END_VAR

		OUT := IN;
		MOVE := IN;
	END_FUNCTION

	FUNCTION MOVE: REAL
		VAR_INPUT
			IN: REAL;
		END_VAR
		VAR_OUTPUT
			OUT: REAL;
		END_VAR

		OUT := IN;
		MOVE := IN;
	END_FUNCTION

	FUNCTION MOVE: LREAL
		VAR_INPUT
			IN: LREAL;
		END_VAR
		VAR_OUTPUT
			OUT: LREAL;
		END_VAR

		OUT := IN;
		MOVE := IN;
	END_FUNCTION

	FUNCTION MOVE: TIME
		VAR_INPUT
			IN: TIME;
		END_VAR
		VAR_OUTPUT
			OUT: TIME;
		END_VAR

		OUT := IN;
		MOVE := IN;
	END_FUNCTION

	FUNCTION MOVE: LTIME
		VAR_INPUT
			IN: LTIME;
		END_VAR
		VAR_OUTPUT
			OUT: LTIME;
		END_VAR

		OUT := IN;
		MOVE := IN;
	END_FUNCTION

	FUNCTION MOVE: STRING[255]
		VAR_INPUT
			IN: STRING[255];
		END_VAR
		VAR_OUTPUT
			OUT: STRING[255];
		END_VAR

		OUT := IN;
		MOVE := IN;
	END_FUNCTION

	FUNCTION MOVE: CHAR
		VAR_INPUT
			IN: CHAR;
		END_VAR
		VAR_OUTPUT
			OUT: CHAR;
		END_VAR

		OUT := IN;
		MOVE := IN;
	END_FUNCTION

	FUNCTION MOVE: DATE
		VAR_INPUT
			IN: DATE;
		END_VAR
		VAR_OUTPUT
			OUT: DATE;
		END_VAR

		OUT := IN;
		MOVE := IN;
	END_FUNCTION

	FUNCTION MOVE: LDATE
		VAR_INPUT
			IN: LDATE;
		END_VAR
		VAR_OUTPUT
			OUT: LDATE;
		END_VAR

		OUT := IN;
		MOVE := IN;
	END_FUNCTION

	FUNCTION MOVE: TOD
		VAR_INPUT
			IN: TOD;
		END_VAR
		VAR_OUTPUT
			OUT: TOD;
		END_VAR

		OUT := IN;
		MOVE := IN;
	END_FUNCTION

	FUNCTION MOVE: LTOD
		VAR_INPUT
			IN: LTOD;
		END_VAR
		VAR_OUTPUT
			OUT: LTOD;
		END_VAR

		OUT := IN;
		MOVE := IN;
	END_FUNCTION

	FUNCTION MOVE: DT
		VAR_INPUT
			IN: DT;
		END_VAR
		VAR_OUTPUT
			OUT: DT;
		END_VAR

		OUT := IN;
		MOVE := IN;
	END_FUNCTION

	FUNCTION MOVE: LDT
		VAR_INPUT
			IN: LDT;
		END_VAR
		VAR_OUTPUT
			OUT: LDT;
		END_VAR

		OUT := IN;
		MOVE := IN;
	END_FUNCTION

	NAMESPACE Test
		USING Std.Unit
		USING Std.Memory
		USING Std.Strings

		{test}
		FUNCTION test_move_int
			VAR
				x: INT := 0;
			END_VAR
			MOVE(42, OUT => x);
			ASSERT_EQ(x, 42);
		END_FUNCTION

		{test}
		FUNCTION test_move_real
			VAR
				x: REAL := 0.0;
			END_VAR
			MOVE(3.14, OUT => x);
			ASSERT_EQ(x, 3.14);
		END_FUNCTION

		{test}
		FUNCTION test_move_bool
			VAR
				x: BOOL := FALSE;
			END_VAR
			MOVE(TRUE, OUT => x);
			ASSERT(x);
		END_FUNCTION

		// --- every overload is independent compiled code: cover the 16 dark
		// ones, each with a boundary value for its type. The i64 lane
		// (LWORD/LINT/ULINT/LREAL/LTIME) is the historically bug-prone path ---

		{test}
		FUNCTION test_move_signed_boundaries
			VAR
				s: SINT;
				d: DINT;
			END_VAR
			MOVE(SINT#-128, OUT => s);
			ASSERT_EQ(s, SINT#-128, 'MOVE SINT at MIN');
			MOVE(DINT#-2147483648, OUT => d);
			ASSERT_EQ(d, DINT#-2147483648, 'MOVE DINT at MIN');
		END_FUNCTION

		{test}
		FUNCTION test_move_unsigned_boundaries
			VAR
				us: USINT;
				u: UINT;
				ud: UDINT;
			END_VAR
			MOVE(USINT#255, OUT => us);
			ASSERT_EQ(us, USINT#255, 'MOVE USINT at MAX');
			MOVE(UINT#65535, OUT => u);
			ASSERT_EQ(u, UINT#65535, 'MOVE UINT at MAX');
			MOVE(UDINT#4294967295, OUT => ud);
			ASSERT_EQ(ud, UDINT#4294967295, 'MOVE UDINT at MAX (above 2^31)');
		END_FUNCTION

		{test}
		FUNCTION test_move_bit_types_sign_bit
			VAR
				b: BYTE;
				w: WORD;
				dw: DWORD;
			END_VAR
			MOVE(BYTE#16#80, OUT => b);
			ASSERT_EQ(b, BYTE#16#80, 'MOVE BYTE with MSB set');
			MOVE(WORD#16#8000, OUT => w);
			ASSERT_EQ(w, WORD#16#8000, 'MOVE WORD with MSB set');
			MOVE(DWORD#16#80000000, OUT => dw);
			ASSERT_EQ(dw, DWORD#16#80000000, 'MOVE DWORD with sign bit set');
		END_FUNCTION

		{test}
		FUNCTION test_move_i64_lane
			VAR
				lw: LWORD;
				li: LINT;
				ul: ULINT;
				lr: LREAL;
			END_VAR
			MOVE(LWORD#16#8000_0000_0000_0000, OUT => lw);
			ASSERT_EQ(lw, LWORD#16#8000_0000_0000_0000, 'MOVE LWORD sign bit');
			MOVE(LINT#-9223372036854775807, OUT => li);
			ASSERT_EQ(li, LINT#-9223372036854775807, 'MOVE LINT near i64 MIN');
			MOVE(ULINT#18446744073709551615, OUT => ul);
			ASSERT_EQ(ul, ULINT#18446744073709551615, 'MOVE ULINT at u64 MAX');
			MOVE(LREAL#1.7976931348623157, OUT => lr);
			ASSERT_EQ(lr, LREAL#1.7976931348623157, 'MOVE LREAL f64 payload');
		END_FUNCTION

		{test}
		FUNCTION test_move_time_types
			VAR
				t: TIME;
				lt: LTIME;
			END_VAR
			MOVE(T#24d20h31m23s647ms, OUT => t);
			ASSERT(t = T#24d20h31m23s647ms, 'MOVE TIME at the signed-ms ceiling');
			MOVE(LTIME#1000d, OUT => lt);
			ASSERT(lt = LTIME#1000d, 'MOVE LTIME on the i64-ns lane');
		END_FUNCTION

		{test}
		FUNCTION test_move_char
			VAR
				c: CHAR;
			END_VAR
			MOVE(CHAR#'z', OUT => c);
			ASSERT_EQ(c, CHAR#'z', 'MOVE CHAR');
		END_FUNCTION

		{test}
		FUNCTION test_move_dates_and_times_of_day
			VAR
				d: DATE;
				ld: LDATE;
				t: TOD;
				lt: LTOD;
				dt1: DT;
				ldt1: LDT;
			END_VAR
			MOVE(D#2024-01-31, OUT => d);
			ASSERT(d = D#2024-01-31, 'MOVE DATE');
			ld := MOVE(LDATE#2024-02-29);
			ASSERT(ld = LDATE#2024-02-29, 'MOVE LDATE');
			MOVE(TOD#12:30:45.123, OUT => t);
			ASSERT(t = TOD#12:30:45.123, 'MOVE TOD');
			lt := MOVE(LTOD#23:59:59.999999999);
			ASSERT(lt = LTOD#23:59:59.999999999, 'MOVE LTOD on the i64-ns lane');
			MOVE(DT#2024-01-31-12:30:45, OUT => dt1);
			ASSERT(dt1 = DT#2024-01-31-12:30:45, 'MOVE DT');
			ldt1 := MOVE(LDT#2024-01-31-12:30:45.5);
			ASSERT(ldt1 = LDT#2024-01-31-12:30:45.5, 'MOVE LDT');
		END_FUNCTION

		{test}
		FUNCTION test_move_string
			VAR
				s: STRING[255];
			END_VAR
			MOVE('edge case', OUT => s);
			ASSERT(LEN(s) = 9, 'MOVE STRING length');
			ASSERT(FIND(s, 'edge case') = 1, 'MOVE STRING content');
		END_FUNCTION

		// Its result is OUT, on each type.
		{test}
		FUNCTION test_move_returns_each_type
			VAR
				b1: BOOL := TRUE;
				b2: BOOL;
				si1: SINT := -5;
				si2: SINT;
				i1: INT := -500;
				i2: INT;
				d1: DINT := -70000;
				d2: DINT;
				l1: LINT := -5000000000;
				l2: LINT;
				us1: USINT := 200;
				us2: USINT;
				u1: UINT := 60000;
				u2: UINT;
				ud1: UDINT := 4000000000;
				ud2: UDINT;
				ul1: ULINT := 18446744073709551615;
				ul2: ULINT;
				by1: BYTE := 16#AB;
				by2: BYTE;
				w1: WORD := 16#ABCD;
				w2: WORD;
				dw1: DWORD := 16#ABCDEF01;
				dw2: DWORD;
				lw1: LWORD := 16#ABCDEF0123456789;
				lw2: LWORD;
				r1: REAL := 1.5;
				r2: REAL;
				lr1: LREAL := 2.5;
				lr2: LREAL;
				t1: TIME := T#3s;
				t2: TIME;
				lt1: LTIME := LTIME#4s;
				lt2: LTIME;
				s1: STRING := 'text';
				s2: STRING;
				c1: CHAR := CHAR#'a';
				c2: CHAR;
			END_VAR
			b2 := MOVE(b1);
			ASSERT(b2);
			si2 := MOVE(si1);
			ASSERT(si2 = -5);
			i2 := MOVE(i1);
			ASSERT(i2 = -500);
			d2 := MOVE(d1);
			ASSERT(d2 = -70000);
			l2 := MOVE(l1);
			ASSERT(l2 = -5000000000);
			us2 := MOVE(us1);
			ASSERT(us2 = 200);
			u2 := MOVE(u1);
			ASSERT(u2 = 60000);
			ud2 := MOVE(ud1);
			ASSERT(ud2 = 4000000000);
			ul2 := MOVE(ul1);
			ASSERT(ul2 = 18446744073709551615);
			by2 := MOVE(by1);
			ASSERT(by2 = 16#AB);
			w2 := MOVE(w1);
			ASSERT(w2 = 16#ABCD);
			dw2 := MOVE(dw1);
			ASSERT(dw2 = 16#ABCDEF01);
			lw2 := MOVE(lw1);
			ASSERT(lw2 = 16#ABCDEF0123456789);
			r2 := MOVE(r1);
			ASSERT(r2 = 1.5);
			lr2 := MOVE(lr1);
			ASSERT(lr2 = 2.5);
			t2 := MOVE(t1);
			ASSERT(t2 = T#3s);
			lt2 := MOVE(lt1);
			ASSERT(lt2 = LTIME#4s);
			s2 := MOVE(s1);
			ASSERT(s2 = 'text');
			c2 := MOVE(c1);
			ASSERT(c2 = CHAR#'a');
		END_FUNCTION

		// A literal takes the type of what it is moved into.
		{test}
		FUNCTION test_move_a_literal
			VAR
				i: INT;
				d: DINT;
				l: LINT;
				u: UINT;
				x: REAL;
				y: LREAL;
				s: STRING;
				b: BOOL;
				w: WORD;
				t: TIME;
			END_VAR
			i := MOVE(5);
			ASSERT(i = 5);
			d := MOVE(70000);
			ASSERT(d = 70000);
			l := MOVE(5000000000);
			ASSERT(l = 5000000000);
			u := MOVE(60000);
			ASSERT(u = 60000);
			x := MOVE(1.5);
			ASSERT(x = 1.5);
			y := MOVE(2.5);
			ASSERT(y = 2.5);
			s := MOVE('abc');
			ASSERT(s = 'abc');
			b := MOVE(TRUE);
			ASSERT(b);
			w := MOVE(WORD#1);
			ASSERT(w = 1);
			t := MOVE(T#1s);
			ASSERT(t = T#1s);
		END_FUNCTION

		// The value widens into a wider target, as any value does.
		{test}
		FUNCTION test_move_into_a_wider_target
			VAR
				si: SINT := -3;
				i: INT := -3;
				d: DINT;
				l: LINT;
				x: REAL;
			END_VAR
			d := MOVE(i);
			ASSERT(d = -3);
			l := MOVE(si);
			ASSERT(l = -3);
			x := MOVE(i);
			ASSERT(x = -3.0);
		END_FUNCTION

		{test}
		FUNCTION test_move_in_an_expression
			VAR
				i: INT := 4;
				b: BOOL := TRUE;
				a: ARRAY[0..4] OF INT;
			END_VAR
			ASSERT(MOVE(i) = 4);
			ASSERT(MOVE(i) + 1 = 5);
			ASSERT(MOVE(MOVE(i)) = 4);
			ASSERT(MOVE(b));
			a[MOVE(i)] := 9;
			ASSERT(a[4] = 9);
			ASSERT(MOVE(a[MOVE(i)]) = 9);
		END_FUNCTION

		// A call may name its output as well.
		{test}
		FUNCTION test_move_returns_what_it_writes
			VAR
				x: INT;
				y: INT;
			END_VAR
			x := MOVE(IN := 6, OUT => y);
			ASSERT(x = 6);
			ASSERT(y = 6);
		END_FUNCTION

		{test}
		FUNCTION test_move_string_past_80_bytes
			VAR
				long: STRING[200] := '01234567890123456789012345678901234567890123456789012345678901234567890123456789012345678901234567890123456789012345678901234567890123456789012345678901234567890123456789012345678901234567890123456789';
				s: STRING[255];
			END_VAR
			MOVE(long, OUT => s);
			ASSERT(LEN(s) = 200, 'MOVE keeps the bytes past 80');
		END_FUNCTION
	END_NAMESPACE
END_NAMESPACE

(* ---- Selection.st ---- *)
/*
Selection functions.

Each has one overload per type it applies to, and returns the type it was
given.
*/
NAMESPACE Std.Selection

	/* Returns `IN0` when `G` is `FALSE`, and `IN1` when it is `TRUE`.

	   # Examples

	   ```iecst
	   n := SEL(TRUE, 10, 42);   // 42
	   n := SEL(FALSE, 10, 42);  // 10
	   ```
	*/
	FUNCTION SEL: BOOL
		VAR_INPUT
			G: BOOL;
			IN0: BOOL;
			IN1: BOOL;
		END_VAR

		IF G THEN
			SEL := IN1;
		ELSE
			SEL := IN0;
		END_IF;
	END_FUNCTION

	FUNCTION SEL: SINT
		VAR_INPUT
			G: BOOL;
			IN0: SINT;
			IN1: SINT;
		END_VAR

		IF G THEN
			SEL := IN1;
		ELSE
			SEL := IN0;
		END_IF;
	END_FUNCTION

	FUNCTION SEL: INT
		VAR_INPUT
			G: BOOL;
			IN0: INT;
			IN1: INT;
		END_VAR

		IF G THEN
			SEL := IN1;
		ELSE
			SEL := IN0;
		END_IF;
	END_FUNCTION

	FUNCTION SEL: DINT
		VAR_INPUT
			G: BOOL;
			IN0: DINT;
			IN1: DINT;
		END_VAR

		IF G THEN
			SEL := IN1;
		ELSE
			SEL := IN0;
		END_IF;
	END_FUNCTION

	FUNCTION SEL: LINT
		VAR_INPUT
			G: BOOL;
			IN0: LINT;
			IN1: LINT;
		END_VAR

		IF G THEN
			SEL := IN1;
		ELSE
			SEL := IN0;
		END_IF;
	END_FUNCTION

	FUNCTION SEL: USINT
		VAR_INPUT
			G: BOOL;
			IN0: USINT;
			IN1: USINT;
		END_VAR

		IF G THEN
			SEL := IN1;
		ELSE
			SEL := IN0;
		END_IF;
	END_FUNCTION

	FUNCTION SEL: UINT
		VAR_INPUT
			G: BOOL;
			IN0: UINT;
			IN1: UINT;
		END_VAR

		IF G THEN
			SEL := IN1;
		ELSE
			SEL := IN0;
		END_IF;
	END_FUNCTION

	FUNCTION SEL: UDINT
		VAR_INPUT
			G: BOOL;
			IN0: UDINT;
			IN1: UDINT;
		END_VAR

		IF G THEN
			SEL := IN1;
		ELSE
			SEL := IN0;
		END_IF;
	END_FUNCTION

	FUNCTION SEL: ULINT
		VAR_INPUT
			G: BOOL;
			IN0: ULINT;
			IN1: ULINT;
		END_VAR

		IF G THEN
			SEL := IN1;
		ELSE
			SEL := IN0;
		END_IF;
	END_FUNCTION

	FUNCTION SEL: BYTE
		VAR_INPUT
			G: BOOL;
			IN0: BYTE;
			IN1: BYTE;
		END_VAR

		IF G THEN
			SEL := IN1;
		ELSE
			SEL := IN0;
		END_IF;
	END_FUNCTION

	FUNCTION SEL: WORD
		VAR_INPUT
			G: BOOL;
			IN0: WORD;
			IN1: WORD;
		END_VAR

		IF G THEN
			SEL := IN1;
		ELSE
			SEL := IN0;
		END_IF;
	END_FUNCTION

	FUNCTION SEL: DWORD
		VAR_INPUT
			G: BOOL;
			IN0: DWORD;
			IN1: DWORD;
		END_VAR

		IF G THEN
			SEL := IN1;
		ELSE
			SEL := IN0;
		END_IF;
	END_FUNCTION

	FUNCTION SEL: LWORD
		VAR_INPUT
			G: BOOL;
			IN0: LWORD;
			IN1: LWORD;
		END_VAR

		IF G THEN
			SEL := IN1;
		ELSE
			SEL := IN0;
		END_IF;
	END_FUNCTION

	FUNCTION SEL: REAL
		VAR_INPUT
			G: BOOL;
			IN0: REAL;
			IN1: REAL;
		END_VAR

		IF G THEN
			SEL := IN1;
		ELSE
			SEL := IN0;
		END_IF;
	END_FUNCTION

	FUNCTION SEL: LREAL
		VAR_INPUT
			G: BOOL;
			IN0: LREAL;
			IN1: LREAL;
		END_VAR

		IF G THEN
			SEL := IN1;
		ELSE
			SEL := IN0;
		END_IF;
	END_FUNCTION

	FUNCTION SEL: TIME
		VAR_INPUT
			G: BOOL;
			IN0: TIME;
			IN1: TIME;
		END_VAR

		IF G THEN
			SEL := IN1;
		ELSE
			SEL := IN0;
		END_IF;
	END_FUNCTION

	FUNCTION SEL: LTIME
		VAR_INPUT
			G: BOOL;
			IN0: LTIME;
			IN1: LTIME;
		END_VAR

		IF G THEN
			SEL := IN1;
		ELSE
			SEL := IN0;
		END_IF;
	END_FUNCTION

	FUNCTION SEL: DATE
		VAR_INPUT
			G: BOOL;
			IN0: DATE;
			IN1: DATE;
		END_VAR

		IF G THEN
			SEL := IN1;
		ELSE
			SEL := IN0;
		END_IF;
	END_FUNCTION

	FUNCTION SEL: LDATE
		VAR_INPUT
			G: BOOL;
			IN0: LDATE;
			IN1: LDATE;
		END_VAR

		IF G THEN
			SEL := IN1;
		ELSE
			SEL := IN0;
		END_IF;
	END_FUNCTION

	FUNCTION SEL: TOD
		VAR_INPUT
			G: BOOL;
			IN0: TOD;
			IN1: TOD;
		END_VAR

		IF G THEN
			SEL := IN1;
		ELSE
			SEL := IN0;
		END_IF;
	END_FUNCTION

	FUNCTION SEL: LTOD
		VAR_INPUT
			G: BOOL;
			IN0: LTOD;
			IN1: LTOD;
		END_VAR

		IF G THEN
			SEL := IN1;
		ELSE
			SEL := IN0;
		END_IF;
	END_FUNCTION

	FUNCTION SEL: DT
		VAR_INPUT
			G: BOOL;
			IN0: DT;
			IN1: DT;
		END_VAR

		IF G THEN
			SEL := IN1;
		ELSE
			SEL := IN0;
		END_IF;
	END_FUNCTION

	FUNCTION SEL: LDT
		VAR_INPUT
			G: BOOL;
			IN0: LDT;
			IN1: LDT;
		END_VAR

		IF G THEN
			SEL := IN1;
		ELSE
			SEL := IN0;
		END_IF;
	END_FUNCTION

	FUNCTION SEL: CHAR
		VAR_INPUT
			G: BOOL;
			IN0: CHAR;
			IN1: CHAR;
		END_VAR

		IF G THEN
			SEL := IN1;
		ELSE
			SEL := IN0;
		END_IF;
	END_FUNCTION

	FUNCTION SEL: STRING[255]
		VAR_INPUT
			G: BOOL;
			IN0: STRING[255];
			IN1: STRING[255];
		END_VAR

		IF G THEN
			SEL := IN1;
		ELSE
			SEL := IN0;
		END_IF;
	END_FUNCTION

	/* Returns `IN` kept within `MN` and `MX`.

	   `MX` wins when `MN` is greater than `MX`.

	   # Examples

	   ```iecst
	   n := LIMIT(0, 15, 10);  // 10
	   n := LIMIT(0, -5, 10);  // 0
	   n := LIMIT(0, 5, 10);   // 5
	   ```
	*/
	FUNCTION LIMIT: BOOL
		VAR_INPUT
			MN: BOOL;
			IN: BOOL;
			MX: BOOL;
		END_VAR

		(* IEC 61131-3 Table 32.5: OUT := MIN(MAX(IN, MN), MX), so MX wins when MN > MX. *)
		LIMIT := IN;
		IF LIMIT < MN THEN
			LIMIT := MN;
		END_IF;
		IF LIMIT > MX THEN
			LIMIT := MX;
		END_IF;
	END_FUNCTION

	FUNCTION LIMIT: SINT
		VAR_INPUT
			MN: SINT;
			IN: SINT;
			MX: SINT;
		END_VAR

		(* IEC 61131-3 Table 32.5: OUT := MIN(MAX(IN, MN), MX), so MX wins when MN > MX. *)
		LIMIT := IN;
		IF LIMIT < MN THEN
			LIMIT := MN;
		END_IF;
		IF LIMIT > MX THEN
			LIMIT := MX;
		END_IF;
	END_FUNCTION

	FUNCTION LIMIT: INT
		VAR_INPUT
			MN: INT;
			IN: INT;
			MX: INT;
		END_VAR

		(* IEC 61131-3 Table 32.5: OUT := MIN(MAX(IN, MN), MX), so MX wins when MN > MX. *)
		LIMIT := IN;
		IF LIMIT < MN THEN
			LIMIT := MN;
		END_IF;
		IF LIMIT > MX THEN
			LIMIT := MX;
		END_IF;
	END_FUNCTION

	FUNCTION LIMIT: DINT
		VAR_INPUT
			MN: DINT;
			IN: DINT;
			MX: DINT;
		END_VAR

		(* IEC 61131-3 Table 32.5: OUT := MIN(MAX(IN, MN), MX), so MX wins when MN > MX. *)
		LIMIT := IN;
		IF LIMIT < MN THEN
			LIMIT := MN;
		END_IF;
		IF LIMIT > MX THEN
			LIMIT := MX;
		END_IF;
	END_FUNCTION

	FUNCTION LIMIT: LINT
		VAR_INPUT
			MN: LINT;
			IN: LINT;
			MX: LINT;
		END_VAR

		(* IEC 61131-3 Table 32.5: OUT := MIN(MAX(IN, MN), MX), so MX wins when MN > MX. *)
		LIMIT := IN;
		IF LIMIT < MN THEN
			LIMIT := MN;
		END_IF;
		IF LIMIT > MX THEN
			LIMIT := MX;
		END_IF;
	END_FUNCTION

	FUNCTION LIMIT: USINT
		VAR_INPUT
			MN: USINT;
			IN: USINT;
			MX: USINT;
		END_VAR

		(* IEC 61131-3 Table 32.5: OUT := MIN(MAX(IN, MN), MX), so MX wins when MN > MX. *)
		LIMIT := IN;
		IF LIMIT < MN THEN
			LIMIT := MN;
		END_IF;
		IF LIMIT > MX THEN
			LIMIT := MX;
		END_IF;
	END_FUNCTION

	FUNCTION LIMIT: UINT
		VAR_INPUT
			MN: UINT;
			IN: UINT;
			MX: UINT;
		END_VAR

		(* IEC 61131-3 Table 32.5: OUT := MIN(MAX(IN, MN), MX), so MX wins when MN > MX. *)
		LIMIT := IN;
		IF LIMIT < MN THEN
			LIMIT := MN;
		END_IF;
		IF LIMIT > MX THEN
			LIMIT := MX;
		END_IF;
	END_FUNCTION

	FUNCTION LIMIT: UDINT
		VAR_INPUT
			MN: UDINT;
			IN: UDINT;
			MX: UDINT;
		END_VAR

		(* IEC 61131-3 Table 32.5: OUT := MIN(MAX(IN, MN), MX), so MX wins when MN > MX. *)
		LIMIT := IN;
		IF LIMIT < MN THEN
			LIMIT := MN;
		END_IF;
		IF LIMIT > MX THEN
			LIMIT := MX;
		END_IF;
	END_FUNCTION

	FUNCTION LIMIT: ULINT
		VAR_INPUT
			MN: ULINT;
			IN: ULINT;
			MX: ULINT;
		END_VAR

		(* IEC 61131-3 Table 32.5: OUT := MIN(MAX(IN, MN), MX), so MX wins when MN > MX. *)
		LIMIT := IN;
		IF LIMIT < MN THEN
			LIMIT := MN;
		END_IF;
		IF LIMIT > MX THEN
			LIMIT := MX;
		END_IF;
	END_FUNCTION

	FUNCTION LIMIT: BYTE
		VAR_INPUT
			MN: BYTE;
			IN: BYTE;
			MX: BYTE;
		END_VAR

		(* IEC 61131-3 Table 32.5: OUT := MIN(MAX(IN, MN), MX), so MX wins when MN > MX. *)
		LIMIT := IN;
		IF LIMIT < MN THEN
			LIMIT := MN;
		END_IF;
		IF LIMIT > MX THEN
			LIMIT := MX;
		END_IF;
	END_FUNCTION

	FUNCTION LIMIT: WORD
		VAR_INPUT
			MN: WORD;
			IN: WORD;
			MX: WORD;
		END_VAR

		(* IEC 61131-3 Table 32.5: OUT := MIN(MAX(IN, MN), MX), so MX wins when MN > MX. *)
		LIMIT := IN;
		IF LIMIT < MN THEN
			LIMIT := MN;
		END_IF;
		IF LIMIT > MX THEN
			LIMIT := MX;
		END_IF;
	END_FUNCTION

	FUNCTION LIMIT: DWORD
		VAR_INPUT
			MN: DWORD;
			IN: DWORD;
			MX: DWORD;
		END_VAR

		(* IEC 61131-3 Table 32.5: OUT := MIN(MAX(IN, MN), MX), so MX wins when MN > MX. *)
		LIMIT := IN;
		IF LIMIT < MN THEN
			LIMIT := MN;
		END_IF;
		IF LIMIT > MX THEN
			LIMIT := MX;
		END_IF;
	END_FUNCTION

	FUNCTION LIMIT: LWORD
		VAR_INPUT
			MN: LWORD;
			IN: LWORD;
			MX: LWORD;
		END_VAR

		(* IEC 61131-3 Table 32.5: OUT := MIN(MAX(IN, MN), MX), so MX wins when MN > MX. *)
		LIMIT := IN;
		IF LIMIT < MN THEN
			LIMIT := MN;
		END_IF;
		IF LIMIT > MX THEN
			LIMIT := MX;
		END_IF;
	END_FUNCTION

	FUNCTION LIMIT: REAL
		VAR_INPUT
			MN: REAL;
			IN: REAL;
			MX: REAL;
		END_VAR

		(* IEC 61131-3 Table 32.5: OUT := MIN(MAX(IN, MN), MX), so MX wins when MN > MX. *)
		LIMIT := IN;
		IF LIMIT < MN THEN
			LIMIT := MN;
		END_IF;
		IF LIMIT > MX THEN
			LIMIT := MX;
		END_IF;
	END_FUNCTION

	FUNCTION LIMIT: LREAL
		VAR_INPUT
			MN: LREAL;
			IN: LREAL;
			MX: LREAL;
		END_VAR

		(* IEC 61131-3 Table 32.5: OUT := MIN(MAX(IN, MN), MX), so MX wins when MN > MX. *)
		LIMIT := IN;
		IF LIMIT < MN THEN
			LIMIT := MN;
		END_IF;
		IF LIMIT > MX THEN
			LIMIT := MX;
		END_IF;
	END_FUNCTION

	FUNCTION LIMIT: TIME
		VAR_INPUT
			MN: TIME;
			IN: TIME;
			MX: TIME;
		END_VAR

		(* IEC 61131-3 Table 32.5: OUT := MIN(MAX(IN, MN), MX), so MX wins when MN > MX. *)
		LIMIT := IN;
		IF LIMIT < MN THEN
			LIMIT := MN;
		END_IF;
		IF LIMIT > MX THEN
			LIMIT := MX;
		END_IF;
	END_FUNCTION

	FUNCTION LIMIT: LTIME
		VAR_INPUT
			MN: LTIME;
			IN: LTIME;
			MX: LTIME;
		END_VAR

		(* IEC 61131-3 Table 32.5: OUT := MIN(MAX(IN, MN), MX), so MX wins when MN > MX. *)
		LIMIT := IN;
		IF LIMIT < MN THEN
			LIMIT := MN;
		END_IF;
		IF LIMIT > MX THEN
			LIMIT := MX;
		END_IF;
	END_FUNCTION

	FUNCTION LIMIT: DATE
		VAR_INPUT
			MN: DATE;
			IN: DATE;
			MX: DATE;
		END_VAR

		(* IEC 61131-3 Table 32.5: OUT := MIN(MAX(IN, MN), MX), so MX wins when MN > MX. *)
		LIMIT := IN;
		IF LIMIT < MN THEN
			LIMIT := MN;
		END_IF;
		IF LIMIT > MX THEN
			LIMIT := MX;
		END_IF;
	END_FUNCTION

	FUNCTION LIMIT: LDATE
		VAR_INPUT
			MN: LDATE;
			IN: LDATE;
			MX: LDATE;
		END_VAR

		(* IEC 61131-3 Table 32.5: OUT := MIN(MAX(IN, MN), MX), so MX wins when MN > MX. *)
		LIMIT := IN;
		IF LIMIT < MN THEN
			LIMIT := MN;
		END_IF;
		IF LIMIT > MX THEN
			LIMIT := MX;
		END_IF;
	END_FUNCTION

	FUNCTION LIMIT: TOD
		VAR_INPUT
			MN: TOD;
			IN: TOD;
			MX: TOD;
		END_VAR

		(* IEC 61131-3 Table 32.5: OUT := MIN(MAX(IN, MN), MX), so MX wins when MN > MX. *)
		LIMIT := IN;
		IF LIMIT < MN THEN
			LIMIT := MN;
		END_IF;
		IF LIMIT > MX THEN
			LIMIT := MX;
		END_IF;
	END_FUNCTION

	FUNCTION LIMIT: LTOD
		VAR_INPUT
			MN: LTOD;
			IN: LTOD;
			MX: LTOD;
		END_VAR

		(* IEC 61131-3 Table 32.5: OUT := MIN(MAX(IN, MN), MX), so MX wins when MN > MX. *)
		LIMIT := IN;
		IF LIMIT < MN THEN
			LIMIT := MN;
		END_IF;
		IF LIMIT > MX THEN
			LIMIT := MX;
		END_IF;
	END_FUNCTION

	FUNCTION LIMIT: DT
		VAR_INPUT
			MN: DT;
			IN: DT;
			MX: DT;
		END_VAR

		(* IEC 61131-3 Table 32.5: OUT := MIN(MAX(IN, MN), MX), so MX wins when MN > MX. *)
		LIMIT := IN;
		IF LIMIT < MN THEN
			LIMIT := MN;
		END_IF;
		IF LIMIT > MX THEN
			LIMIT := MX;
		END_IF;
	END_FUNCTION

	FUNCTION LIMIT: LDT
		VAR_INPUT
			MN: LDT;
			IN: LDT;
			MX: LDT;
		END_VAR

		(* IEC 61131-3 Table 32.5: OUT := MIN(MAX(IN, MN), MX), so MX wins when MN > MX. *)
		LIMIT := IN;
		IF LIMIT < MN THEN
			LIMIT := MN;
		END_IF;
		IF LIMIT > MX THEN
			LIMIT := MX;
		END_IF;
	END_FUNCTION

	FUNCTION LIMIT: CHAR
		VAR_INPUT
			MN: CHAR;
			IN: CHAR;
			MX: CHAR;
		END_VAR

		(* IEC 61131-3 Table 32.5: OUT := MIN(MAX(IN, MN), MX), so MX wins when MN > MX. *)
		LIMIT := IN;
		IF LIMIT < MN THEN
			LIMIT := MN;
		END_IF;
		IF LIMIT > MX THEN
			LIMIT := MX;
		END_IF;
	END_FUNCTION

	FUNCTION LIMIT: STRING[255]
		VAR_INPUT
			MN: STRING[255];
			IN: STRING[255];
			MX: STRING[255];
		END_VAR

		(* IEC 61131-3 Table 32.5: OUT := MIN(MAX(IN, MN), MX), so MX wins when MN > MX. *)
		LIMIT := IN;
		IF LIMIT < MN THEN
			LIMIT := MN;
		END_IF;
		IF LIMIT > MX THEN
			LIMIT := MX;
		END_IF;
	END_FUNCTION

	/* Returns the smallest of its inputs, however many there are.

	   A `STRING` takes two, three or four.

	   # Examples

	   ```iecst
	   n := MIN(3, 5);     // 3
	   n := MIN(7, 9, 4);  // 4
	   ```
	*/
	FUNCTION MIN: BOOL
		VAR_INPUT
			IN: BOOL...;
		END_VAR

		MIN := ...IN MIN;
	END_FUNCTION

	FUNCTION MIN: SINT
		VAR_INPUT
			IN: SINT...;
		END_VAR

		MIN := ...IN MIN;
	END_FUNCTION

	FUNCTION MIN: INT
		VAR_INPUT
			IN: INT...;
		END_VAR

		MIN := ...IN MIN;
	END_FUNCTION

	FUNCTION MIN: DINT
		VAR_INPUT
			IN: DINT...;
		END_VAR

		MIN := ...IN MIN;
	END_FUNCTION

	FUNCTION MIN: LINT
		VAR_INPUT
			IN: LINT...;
		END_VAR

		MIN := ...IN MIN;
	END_FUNCTION

	FUNCTION MIN: USINT
		VAR_INPUT
			IN: USINT...;
		END_VAR

		MIN := ...IN MIN;
	END_FUNCTION

	FUNCTION MIN: UINT
		VAR_INPUT
			IN: UINT...;
		END_VAR

		MIN := ...IN MIN;
	END_FUNCTION

	FUNCTION MIN: UDINT
		VAR_INPUT
			IN: UDINT...;
		END_VAR

		MIN := ...IN MIN;
	END_FUNCTION

	FUNCTION MIN: ULINT
		VAR_INPUT
			IN: ULINT...;
		END_VAR

		MIN := ...IN MIN;
	END_FUNCTION

	FUNCTION MIN: BYTE
		VAR_INPUT
			IN: BYTE...;
		END_VAR

		MIN := ...IN MIN;
	END_FUNCTION

	FUNCTION MIN: WORD
		VAR_INPUT
			IN: WORD...;
		END_VAR

		MIN := ...IN MIN;
	END_FUNCTION

	FUNCTION MIN: DWORD
		VAR_INPUT
			IN: DWORD...;
		END_VAR

		MIN := ...IN MIN;
	END_FUNCTION

	FUNCTION MIN: LWORD
		VAR_INPUT
			IN: LWORD...;
		END_VAR

		MIN := ...IN MIN;
	END_FUNCTION

	FUNCTION MIN: REAL
		VAR_INPUT
			IN: REAL...;
		END_VAR

		MIN := ...IN MIN;
	END_FUNCTION

	FUNCTION MIN: LREAL
		VAR_INPUT
			IN: LREAL...;
		END_VAR

		MIN := ...IN MIN;
	END_FUNCTION

	FUNCTION MIN: STRING[255]
		VAR_INPUT
			IN1: STRING[255];
			IN2: STRING[255];
		END_VAR

		MIN := IN1;
		IF IN2 < MIN THEN
			MIN := IN2;
		END_IF;
	END_FUNCTION

	FUNCTION MIN: STRING[255]
		VAR_INPUT
			IN1: STRING[255];
			IN2: STRING[255];
			IN3: STRING[255];
		END_VAR

		MIN := IN1;
		IF IN2 < MIN THEN
			MIN := IN2;
		END_IF;
		IF IN3 < MIN THEN
			MIN := IN3;
		END_IF;
	END_FUNCTION

	FUNCTION MIN: STRING[255]
		VAR_INPUT
			IN1: STRING[255];
			IN2: STRING[255];
			IN3: STRING[255];
			IN4: STRING[255];
		END_VAR

		MIN := IN1;
		IF IN2 < MIN THEN
			MIN := IN2;
		END_IF;
		IF IN3 < MIN THEN
			MIN := IN3;
		END_IF;
		IF IN4 < MIN THEN
			MIN := IN4;
		END_IF;
	END_FUNCTION

	FUNCTION MIN: TIME
		VAR_INPUT
			IN: TIME...;
		END_VAR

		MIN := ...IN MIN;
	END_FUNCTION

	FUNCTION MIN: LTIME
		VAR_INPUT
			IN: LTIME...;
		END_VAR

		MIN := ...IN MIN;
	END_FUNCTION

	FUNCTION MIN: DATE
		VAR_INPUT
			IN: DATE...;
		END_VAR

		MIN := ...IN MIN;
	END_FUNCTION

	FUNCTION MIN: LDATE
		VAR_INPUT
			IN: LDATE...;
		END_VAR

		MIN := ...IN MIN;
	END_FUNCTION

	FUNCTION MIN: TOD
		VAR_INPUT
			IN: TOD...;
		END_VAR

		MIN := ...IN MIN;
	END_FUNCTION

	FUNCTION MIN: LTOD
		VAR_INPUT
			IN: LTOD...;
		END_VAR

		MIN := ...IN MIN;
	END_FUNCTION

	FUNCTION MIN: DT
		VAR_INPUT
			IN: DT...;
		END_VAR

		MIN := ...IN MIN;
	END_FUNCTION

	FUNCTION MIN: LDT
		VAR_INPUT
			IN: LDT...;
		END_VAR

		MIN := ...IN MIN;
	END_FUNCTION

	FUNCTION MIN: CHAR
		VAR_INPUT
			IN: CHAR...;
		END_VAR

		MIN := ...IN MIN;
	END_FUNCTION

	/* Returns the largest of its inputs, however many there are.

	   A `STRING` takes two, three or four.

	   # Examples

	   ```iecst
	   n := MAX(3, 5);     // 5
	   n := MAX(7, 9, 4);  // 9
	   ```
	*/
	FUNCTION MAX: BOOL
		VAR_INPUT
			IN: BOOL...;
		END_VAR

		MAX := ...IN MAX;
	END_FUNCTION

	FUNCTION MAX: SINT
		VAR_INPUT
			IN: SINT...;
		END_VAR

		MAX := ...IN MAX;
	END_FUNCTION

	FUNCTION MAX: INT
		VAR_INPUT
			IN: INT...;
		END_VAR

		MAX := ...IN MAX;
	END_FUNCTION

	FUNCTION MAX: DINT
		VAR_INPUT
			IN: DINT...;
		END_VAR

		MAX := ...IN MAX;
	END_FUNCTION

	FUNCTION MAX: LINT
		VAR_INPUT
			IN: LINT...;
		END_VAR

		MAX := ...IN MAX;
	END_FUNCTION

	FUNCTION MAX: USINT
		VAR_INPUT
			IN: USINT...;
		END_VAR

		MAX := ...IN MAX;
	END_FUNCTION

	FUNCTION MAX: UINT
		VAR_INPUT
			IN: UINT...;
		END_VAR

		MAX := ...IN MAX;
	END_FUNCTION

	FUNCTION MAX: UDINT
		VAR_INPUT
			IN: UDINT...;
		END_VAR

		MAX := ...IN MAX;
	END_FUNCTION

	FUNCTION MAX: ULINT
		VAR_INPUT
			IN: ULINT...;
		END_VAR

		MAX := ...IN MAX;
	END_FUNCTION

	FUNCTION MAX: BYTE
		VAR_INPUT
			IN: BYTE...;
		END_VAR

		MAX := ...IN MAX;
	END_FUNCTION

	FUNCTION MAX: WORD
		VAR_INPUT
			IN: WORD...;
		END_VAR

		MAX := ...IN MAX;
	END_FUNCTION

	FUNCTION MAX: DWORD
		VAR_INPUT
			IN: DWORD...;
		END_VAR

		MAX := ...IN MAX;
	END_FUNCTION

	FUNCTION MAX: LWORD
		VAR_INPUT
			IN: LWORD...;
		END_VAR

		MAX := ...IN MAX;
	END_FUNCTION

	FUNCTION MAX: REAL
		VAR_INPUT
			IN: REAL...;
		END_VAR

		MAX := ...IN MAX;
	END_FUNCTION

	FUNCTION MAX: LREAL
		VAR_INPUT
			IN: LREAL...;
		END_VAR

		MAX := ...IN MAX;
	END_FUNCTION

	FUNCTION MAX: STRING[255]
		VAR_INPUT
			IN1: STRING[255];
			IN2: STRING[255];
		END_VAR

		MAX := IN1;
		IF IN2 > MAX THEN
			MAX := IN2;
		END_IF;
	END_FUNCTION

	FUNCTION MAX: STRING[255]
		VAR_INPUT
			IN1: STRING[255];
			IN2: STRING[255];
			IN3: STRING[255];
		END_VAR

		MAX := IN1;
		IF IN2 > MAX THEN
			MAX := IN2;
		END_IF;
		IF IN3 > MAX THEN
			MAX := IN3;
		END_IF;
	END_FUNCTION

	FUNCTION MAX: STRING[255]
		VAR_INPUT
			IN1: STRING[255];
			IN2: STRING[255];
			IN3: STRING[255];
			IN4: STRING[255];
		END_VAR

		MAX := IN1;
		IF IN2 > MAX THEN
			MAX := IN2;
		END_IF;
		IF IN3 > MAX THEN
			MAX := IN3;
		END_IF;
		IF IN4 > MAX THEN
			MAX := IN4;
		END_IF;
	END_FUNCTION

	FUNCTION MAX: TIME
		VAR_INPUT
			IN: TIME...;
		END_VAR

		MAX := ...IN MAX;
	END_FUNCTION

	FUNCTION MAX: LTIME
		VAR_INPUT
			IN: LTIME...;
		END_VAR

		MAX := ...IN MAX;
	END_FUNCTION

	FUNCTION MAX: DATE
		VAR_INPUT
			IN: DATE...;
		END_VAR

		MAX := ...IN MAX;
	END_FUNCTION

	FUNCTION MAX: LDATE
		VAR_INPUT
			IN: LDATE...;
		END_VAR

		MAX := ...IN MAX;
	END_FUNCTION

	FUNCTION MAX: TOD
		VAR_INPUT
			IN: TOD...;
		END_VAR

		MAX := ...IN MAX;
	END_FUNCTION

	FUNCTION MAX: LTOD
		VAR_INPUT
			IN: LTOD...;
		END_VAR

		MAX := ...IN MAX;
	END_FUNCTION

	FUNCTION MAX: DT
		VAR_INPUT
			IN: DT...;
		END_VAR

		MAX := ...IN MAX;
	END_FUNCTION

	FUNCTION MAX: LDT
		VAR_INPUT
			IN: LDT...;
		END_VAR

		MAX := ...IN MAX;
	END_FUNCTION

	FUNCTION MAX: CHAR
		VAR_INPUT
			IN: CHAR...;
		END_VAR

		MAX := ...IN MAX;
	END_FUNCTION

	/* Returns the input that `K` selects, counting from 0.

	   A `K` below 0 selects the first input, and a `K` past the last selects the
	   last. Every elementary type takes any number of inputs, except `STRING`,
	   which takes two, three or four.

	   `K` is any integer type but `ULINT`. Convert a `ULINT` or a bit string first,
	   with [Std.Convert.ULINT_TO_LINT] or [Std.Convert.WORD_TO_LINT].

	   # Examples

	   ```iecst
	   n := MUX(1, 10, 20, 30);   // 20
	   n := MUX(-1, 10, 20, 30);  // 10
	   n := MUX(9, 10, 20, 30);   // 30
	   ```
	*/
	FUNCTION MUX: BOOL
		VAR_INPUT
			K: LINT;
			IN: BOOL...;
		END_VAR

		MUX := ...IN[K];
	END_FUNCTION

	FUNCTION MUX: SINT
		VAR_INPUT
			K: LINT;
			IN: SINT...;
		END_VAR

		MUX := ...IN[K];
	END_FUNCTION

	FUNCTION MUX: INT
		VAR_INPUT
			K: LINT;
			IN: INT...;
		END_VAR

		MUX := ...IN[K];
	END_FUNCTION

	FUNCTION MUX: DINT
		VAR_INPUT
			K: LINT;
			IN: DINT...;
		END_VAR

		MUX := ...IN[K];
	END_FUNCTION

	FUNCTION MUX: LINT
		VAR_INPUT
			K: LINT;
			IN: LINT...;
		END_VAR

		MUX := ...IN[K];
	END_FUNCTION

	FUNCTION MUX: USINT
		VAR_INPUT
			K: LINT;
			IN: USINT...;
		END_VAR

		MUX := ...IN[K];
	END_FUNCTION

	FUNCTION MUX: UINT
		VAR_INPUT
			K: LINT;
			IN: UINT...;
		END_VAR

		MUX := ...IN[K];
	END_FUNCTION

	FUNCTION MUX: UDINT
		VAR_INPUT
			K: LINT;
			IN: UDINT...;
		END_VAR

		MUX := ...IN[K];
	END_FUNCTION

	FUNCTION MUX: ULINT
		VAR_INPUT
			K: LINT;
			IN: ULINT...;
		END_VAR

		MUX := ...IN[K];
	END_FUNCTION

	FUNCTION MUX: BYTE
		VAR_INPUT
			K: LINT;
			IN: BYTE...;
		END_VAR

		MUX := ...IN[K];
	END_FUNCTION

	FUNCTION MUX: WORD
		VAR_INPUT
			K: LINT;
			IN: WORD...;
		END_VAR

		MUX := ...IN[K];
	END_FUNCTION

	FUNCTION MUX: DWORD
		VAR_INPUT
			K: LINT;
			IN: DWORD...;
		END_VAR

		MUX := ...IN[K];
	END_FUNCTION

	FUNCTION MUX: LWORD
		VAR_INPUT
			K: LINT;
			IN: LWORD...;
		END_VAR

		MUX := ...IN[K];
	END_FUNCTION

	FUNCTION MUX: REAL
		VAR_INPUT
			K: LINT;
			IN: REAL...;
		END_VAR

		MUX := ...IN[K];
	END_FUNCTION

	FUNCTION MUX: LREAL
		VAR_INPUT
			K: LINT;
			IN: LREAL...;
		END_VAR

		MUX := ...IN[K];
	END_FUNCTION

	FUNCTION MUX: STRING[255]
		VAR_INPUT
			K: LINT;
			IN0: STRING[255];
			IN1: STRING[255];
		END_VAR

		IF K <= 0 THEN
			MUX := IN0;
		ELSE
			MUX := IN1;
		END_IF;
	END_FUNCTION

	FUNCTION MUX: STRING[255]
		VAR_INPUT
			K: LINT;
			IN0: STRING[255];
			IN1: STRING[255];
			IN2: STRING[255];
		END_VAR

		IF K <= 0 THEN
			MUX := IN0;
		ELSIF K = 1 THEN
			MUX := IN1;
		ELSE
			MUX := IN2;
		END_IF;
	END_FUNCTION

	FUNCTION MUX: STRING[255]
		VAR_INPUT
			K: LINT;
			IN0: STRING[255];
			IN1: STRING[255];
			IN2: STRING[255];
			IN3: STRING[255];
		END_VAR

		IF K <= 0 THEN
			MUX := IN0;
		ELSIF K = 1 THEN
			MUX := IN1;
		ELSIF K = 2 THEN
			MUX := IN2;
		ELSE
			MUX := IN3;
		END_IF;
	END_FUNCTION

	FUNCTION MUX: TIME
		VAR_INPUT
			K: LINT;
			IN: TIME...;
		END_VAR

		MUX := ...IN[K];
	END_FUNCTION

	FUNCTION MUX: LTIME
		VAR_INPUT
			K: LINT;
			IN: LTIME...;
		END_VAR

		MUX := ...IN[K];
	END_FUNCTION

	FUNCTION MUX: DATE
		VAR_INPUT
			K: LINT;
			IN: DATE...;
		END_VAR

		MUX := ...IN[K];
	END_FUNCTION

	FUNCTION MUX: LDATE
		VAR_INPUT
			K: LINT;
			IN: LDATE...;
		END_VAR

		MUX := ...IN[K];
	END_FUNCTION

	FUNCTION MUX: TOD
		VAR_INPUT
			K: LINT;
			IN: TOD...;
		END_VAR

		MUX := ...IN[K];
	END_FUNCTION

	FUNCTION MUX: LTOD
		VAR_INPUT
			K: LINT;
			IN: LTOD...;
		END_VAR

		MUX := ...IN[K];
	END_FUNCTION

	FUNCTION MUX: DT
		VAR_INPUT
			K: LINT;
			IN: DT...;
		END_VAR

		MUX := ...IN[K];
	END_FUNCTION

	FUNCTION MUX: LDT
		VAR_INPUT
			K: LINT;
			IN: LDT...;
		END_VAR

		MUX := ...IN[K];
	END_FUNCTION

	FUNCTION MUX: CHAR
		VAR_INPUT
			K: LINT;
			IN: CHAR...;
		END_VAR

		MUX := ...IN[K];
	END_FUNCTION

	NAMESPACE Test
		USING Std.Unit
		USING Std.Selection

		// SEL tests

		{test}
		FUNCTION test_sel_true_returns_in1 ASSERT_EQ(SEL(TRUE, 10, 42), 42);
		END_FUNCTION

		{test}
		FUNCTION test_sel_false_returns_in0 ASSERT_EQ(SEL(FALSE, 10, 42), 10);
		END_FUNCTION

		{test}
		FUNCTION test_sel_real_true ASSERT_EQ(SEL(TRUE, 1.0, 3.14), 3.14);
		END_FUNCTION

		{test}
		FUNCTION test_sel_real_false ASSERT_EQ(SEL(FALSE, 1.0, 3.14), 1.0);
		END_FUNCTION

		// LIMIT tests

		{test}
		FUNCTION test_limit_in_range ASSERT_EQ(LIMIT(0, 5, 10), 5);
		END_FUNCTION

		{test}
		FUNCTION test_limit_below_min ASSERT_EQ(LIMIT(0, -5, 10), 0);
		END_FUNCTION

		{test}
		FUNCTION test_limit_above_max ASSERT_EQ(LIMIT(0, 15, 10), 10);
		END_FUNCTION

		{test}
		FUNCTION test_limit_at_min ASSERT_EQ(LIMIT(0, 0, 10), 0);
		END_FUNCTION

		{test}
		FUNCTION test_limit_at_max ASSERT_EQ(LIMIT(0, 10, 10), 10);
		END_FUNCTION

		{test}
		FUNCTION test_limit_real_clamp_low ASSERT_EQ(LIMIT(0.0, -1.5, 10.0), 0.0);
		END_FUNCTION

		{test}
		FUNCTION test_limit_real_clamp_high ASSERT_EQ(LIMIT(0.0, 15.5, 10.0), 10.0);
		END_FUNCTION

		{test}
		FUNCTION test_limit_real_in_range ASSERT_EQ(LIMIT(0.0, 5.5, 10.0), 5.5);
		END_FUNCTION

		// --- nonzero-MN clamps: a LIMIT body that never assigns its result
		// would return the zero-initialized local and still pass every
		// clamp-low test above. Pin clamps whose expected value is NOT 0 ---

		{test}
		FUNCTION test_limit_nonzero_mn_clamp
			ASSERT_EQ(LIMIT(INT#20, INT#5, INT#30), INT#20, 'clamp low to a nonzero MN');
			ASSERT_EQ(LIMIT(INT#-30, INT#-50, INT#-10), INT#-30, 'negative bounds clamp low');
			ASSERT_EQ(LIMIT(INT#-30, INT#0, INT#-10), INT#-10, 'negative bounds clamp high');
		END_FUNCTION

		// IEC 61131-3 Table 32.5: OUT := MIN(MAX(IN, MN), MX). With the
		// degenerate MN > MX, applying MX last means MX wins.
		{test}
		FUNCTION test_limit_mn_greater_than_mx
			ASSERT_EQ(LIMIT(INT#10, INT#5, INT#0), INT#0, 'MX wins when MN > MX');
		END_FUNCTION

		// --- typed overload coverage: each overload is independent compiled
		// code; the untyped-literal tests above only ever reach INT/REAL ---

		{test}
		FUNCTION test_limit_lint_i64_lane
			ASSERT_EQ(LIMIT(LINT#-5000000000, LINT#-6000000000, LINT#5000000000), LINT#-5000000000, 'i64 clamp low beyond i32 range');
			ASSERT_EQ(LIMIT(LINT#0, LINT#6000000000, LINT#5000000000), LINT#5000000000, 'i64 clamp high beyond i32 range');
		END_FUNCTION

		{test}
		FUNCTION test_limit_udint_above_signed_max
			ASSERT_EQ(LIMIT(UDINT#0, UDINT#4000000000, UDINT#3000000000), UDINT#3000000000, 'unsigned compare above 2^31 must not go signed');
		END_FUNCTION

		{test}
		FUNCTION test_limit_sint_boundaries
			ASSERT_EQ(LIMIT(SINT#-128, SINT#-128, SINT#127), SINT#-128, 'SINT MIN passes through');
			ASSERT_EQ(LIMIT(SINT#-100, SINT#127, SINT#100), SINT#100, 'SINT clamp high');
		END_FUNCTION

		{test}
		FUNCTION test_limit_time
			ASSERT(LIMIT(T#1s, T#500ms, T#10s) = T#1s, 'TIME clamp low');
			ASSERT(LIMIT(T#1s, T#20s, T#10s) = T#10s, 'TIME clamp high');
		END_FUNCTION

		{test}
		FUNCTION test_sel_byte
			ASSERT_EQ(SEL(FALSE, BYTE#16#AA, BYTE#16#55), BYTE#16#AA, 'SEL BYTE G=FALSE');
			ASSERT_EQ(SEL(TRUE, BYTE#16#AA, BYTE#16#55), BYTE#16#55, 'SEL BYTE G=TRUE');
		END_FUNCTION

		{test}
		FUNCTION test_sel_lword_i64_lane
			ASSERT_EQ(SEL(TRUE, LWORD#1, LWORD#16#8000_0000_0000_0000), LWORD#16#8000_0000_0000_0000, 'SEL LWORD picks a sign-bit i64 value');
		END_FUNCTION

		{test}
		FUNCTION test_sel_lint_boundaries
			ASSERT_EQ(SEL(FALSE, LINT#-9223372036854775807, LINT#0), LINT#-9223372036854775807, 'SEL LINT near i64 MIN');
		END_FUNCTION

		{test}
		FUNCTION test_sel_time
			ASSERT(SEL(TRUE, T#1s, T#2s) = T#2s, 'SEL TIME');
		END_FUNCTION

		{test}
		FUNCTION test_sel_bool
			ASSERT_EQ(SEL(TRUE, FALSE, TRUE), TRUE, 'SEL BOOL both branches distinct');
			ASSERT_EQ(SEL(FALSE, FALSE, TRUE), FALSE, 'SEL BOOL G=FALSE');
		END_FUNCTION

		// -- MIN / MAX ------------------------------------------------

		{test}
		FUNCTION test_min_max_int
			ASSERT_EQ(MIN(3, 5), 3);
			ASSERT_EQ(MAX(3, 5), 5);
			ASSERT_EQ(MIN(-2, 2), -2);
			ASSERT_EQ(MAX(-2, 2), 2);
		END_FUNCTION

		{test}
		FUNCTION test_min_max_real
			ASSERT_EQ(MIN(1.5, 2.5), 1.5);
			ASSERT_EQ(MAX(1.5, 2.5), 2.5);
		END_FUNCTION

		{test}
		FUNCTION test_min_max_time
			ASSERT_EQ(MIN(T#1s, T#2s), T#1s);
			ASSERT_EQ(MAX(T#1s, T#2s), T#2s);
		END_FUNCTION

		{test}
		FUNCTION test_min_max_any_number_of_inputs
			ASSERT_EQ(MIN(5), 5);
			ASSERT_EQ(MAX(5), 5);
			ASSERT_EQ(MIN(3, 1, 2), 1);
			ASSERT_EQ(MAX(1, 3, 2), 3);
			ASSERT_EQ(MIN(8, 6, 7, 5, 3, 0, 9), 0);
			ASSERT_EQ(MAX(8, 6, 7, 5, 3, 0, 9), 9);
		END_FUNCTION

		{test}
		FUNCTION test_min_max_widen_to_the_wider_type
			VAR
				i: INT := 1;
				d: DINT := 70000;
				r: REAL := 2.5;
			END_VAR
			ASSERT_EQ(MAX(i, d), DINT#70000);
			ASSERT_EQ(MIN(d, i, d), DINT#1);
			ASSERT_EQ(MIN(i, r), REAL#1.0);
		END_FUNCTION

		{test}
		FUNCTION test_min_max_nest
			ASSERT_EQ(MIN(7, MIN(9, 4)), 4);
			ASSERT_EQ(MAX(7, MAX(9, 4)), 9);
		END_FUNCTION

		// -- MUX ------------------------------------------------------

		{test}
		FUNCTION test_mux_selects
			ASSERT_EQ(MUX(0, 10, 20), 10);
			ASSERT_EQ(MUX(1, 10, 20), 20);
			ASSERT_EQ(MUX(1, 10, 20, 30), 20);
			ASSERT_EQ(MUX(2, 10, 20, 30), 30);
			ASSERT_EQ(MUX(3, 10, 20, 30, 40), 40);
		END_FUNCTION

		{test}
		FUNCTION test_mux_any_number_of_inputs
			ASSERT_EQ(MUX(0, 10), 10);
			ASSERT_EQ(MUX(5, 10, 20, 30, 40, 50, 60, 70), 60);
		END_FUNCTION

		{test}
		FUNCTION test_mux_clamps
			ASSERT_EQ(MUX(-1, 10, 20, 30), 10);
			ASSERT_EQ(MUX(9, 10, 20, 30), 30);
		END_FUNCTION

		{test}
		FUNCTION test_mux_string
			VAR
				s: STRING;
			END_VAR
			s := MUX(1, 'low', 'high');
			ASSERT_EQ(s, 'high');
		END_FUNCTION
	END_NAMESPACE
END_NAMESPACE
